LIN {X 0,Y 115.598,Z 257.735,A -85,B 0,C 180,E1 -25782.895,E2 -25782.895} C_VEL
LIN {X 0,Y 117.67,Z 260.063,A -85,B 0,C 180,E1 -25784.586,E2 -25784.586} C_VEL
LIN {X 0,Y 118.631,Z 260.945,A -85,B 0,C 180,E1 -25785.308,E2 -25785.308} C_VEL
LIN {X 0,Y 120.566,Z 264.086,A -85,B 0,C 180,E1 -25786.824,E2 -25786.824} C_VEL
LIN {X 0,Y 122.311,Z 266.016,A -85,B 0,C 180,E1 -25788.026,E2 -25788.026} C_VEL
LIN {X 0,Y 125.956,Z 271.384,A -85,B 0,C 180,E1 -25790.457,E2 -25790.457} C_VEL
LIN {X 0,Y 130.306,Z 277.986,A -85,B 0,C 180,E1 -25793.063,E2 -25793.063} C_VEL
LIN {X 0,Y 136.455,Z 288.82,A -85,B 0,C 180,E1 -25796.428,E2 -25796.428} C_VEL
LIN {X 0,Y 142.566,Z 302.152,A -85,B 0,C 180,E1 -25799.513,E2 -25799.513} C_VEL
LIN {X 0,Y 139.129,Z 349.924,A -85,B 0,C 180,E1 -25801.622,E2 -25801.622} C_VEL
LIN {X 0,Y 137.337,Z 363.693,A -85,B 0,C 180,E1 -25802.791,E2 -25802.791} C_VEL
LIN {X 0,Y 135.158,Z 375.917,A -85,B 0,C 180,E1 -25804.399,E2 -25804.399} C_VEL
LIN {X 0,Y 132.259,Z 387.767,A -85,B 0,C 180,E1 -25806.521,E2 -25806.521} C_VEL
LIN {X 0,Y 128.943,Z 399.162,A -85,B 0,C 180,E1 -25809.258,E2 -25809.258} C_VEL
LIN {X 0,Y 125.816,Z 408.801,A -85,B 0,C 180,E1 -25812.288,E2 -25812.288} C_VEL
LIN {X 0,Y 122.59,Z 417.663,A -85,B 0,C 180,E1 -25815.82,E2 -25815.82} C_VEL
LIN {X 0,Y 118.993,Z 426.966,A -85,B 0,C 180,E1 -25820.659,E2 -25820.659} C_VEL
LIN {X 0,Y 116.23,Z 434.328,A -85,B 0,C 180,E1 -25825.672,E2 -25825.672} C_VEL
LIN {X 0,Y 114.556,Z 439.301,A -85,B 0,C 180,E1 -25830.006,E2 -25830.006} C_VEL
LIN {X 0,Y 113.016,Z 444.479,A -85,B 0,C 180,E1 -25835.755,E2 -25835.755} C_VEL
LIN {X 0,Y 112.2,Z 447.894,A -85,B 0,C 180,E1 -25840.836,E2 -25840.836} C_VEL
LIN {X 0,Y 112.013,Z 449.826,A -85,B 0,C 180,E1 -25844.54,E2 -25844.54} C_VEL
LIN {X 0,Y 112.506,Z 451.951,A -85,B 0,C 180,E1 -25850.447,E2 -25850.447} C_VEL
LIN {X 0,Y 113.673,Z 452.945,A -85,B 0,C 180,E1 -25855.649,E2 -25855.649} C_VEL
LIN {X 0,Y 116.312,Z 452.961,A -85,B 0,C 180,E1 -25862.23,E2 -25862.23} C_VEL
LIN {X 0,Y 118.692,Z 452.233,A -85,B 0,C 180,E1 -25866.311,E2 -25866.311} C_VEL
LIN {X 0,Y 123.419,Z 449.925,A -85,B 0,C 180,E1 -25872.247,E2 -25872.247} C_VEL
LIN {X 0,Y 128.871,Z 446.362,A -85,B 0,C 180,E1 -25877.413,E2 -25877.413} C_VEL
LIN {X 0,Y 134.492,Z 441.991,A -85,B 0,C 180,E1 -25881.615,E2 -25881.615} C_VEL
LIN {X 0,Y 140.722,Z 436.325,A -85,B 0,C 180,E1 -25885.493,E2 -25885.493} C_VEL
LIN {X 0,Y 147.535,Z 429.154,A -85,B 0,C 180,E1 -25889.032,E2 -25889.032} C_VEL
LIN {X 0,Y 154.85,Z 420.055,A -85,B 0,C 180,E1 -25892.254,E2 -25892.254} C_VEL
LIN {X 0,Y 161.376,Z 410.613,A -85,B 0,C 180,E1 -25894.678,E2 -25894.678} C_VEL
LIN {X 0,Y 167.361,Z 400.08,A -85,B 0,C 180,E1 -25896.72,E2 -25896.72} C_VEL
LIN {X 0,Y 172.914,Z 387.981,A -85,B 0,C 180,E1 -25898.493,E2 -25898.493} C_VEL
LIN {X 0,Y 176.998,Z 376.677,A -85,B 0,C 180,E1 -25899.727,E2 -25899.727} C_VEL
LIN {X 0,Y 180.453,Z 363.897,A -85,B 0,C 180,E1 -25900.713,E2 -25900.713} C_VEL
LIN {X 0,Y 182.767,Z 351.132,A -85,B 0,C 180,E1 -25901.395,E2 -25901.395} C_VEL
LIN {X 0,Y 184.15,Z 337.384,A -85,B 0,C 180,E1 -25901.89,E2 -25901.89} C_VEL
LIN {X 0,Y 180.509,Z 329.961,A -85,B 0,C 180,E1 -25905.125,E2 -25905.125} C_VEL
LIN {X 0,Y 177.491,Z 324.525,A -85,B 0,C 180,E1 -25908.22,E2 -25908.22} C_VEL
LIN {X 0,Y 175.588,Z 321.158,A -85,B 0,C 180,E1 -25910.497,E2 -25910.497} C_VEL
LIN {X 0,Y 173.971,Z 318.349,A -85,B 0,C 180,E1 -25912.748,E2 -25912.748} C_VEL
LIN {X 0,Y 172.019,Z 314.67,A -85,B 0,C 180,E1 -25916.245,E2 -25916.245} C_VEL
LIN {X 0,Y 170.224,Z 311.982,A -85,B 0,C 180,E1 -25920.807,E2 -25920.807} C_VEL
LIN {X 0,Y 169.821,Z 310.313,A -85,B 0,C 180,E1 -25922.93,E2 -25922.93} C_VEL
LIN {X 0,Y 169.608,Z 310.274,A -85,B 0,C 180,E1 -25930.406,E2 -25930.406} C_VEL
LIN {X 0,Y 171.721,Z 314.762,A -85,B 0,C 180,E1 -25937.684,E2 -25937.684} C_VEL
LIN {X 0,Y 172.317,Z 315.843,A -85,B 0,C 180,E1 -25938.909,E2 -25938.909} C_VEL
LIN {X 0,Y 174.722,Z 321.19,A -85,B 0,C 180,E1 -25942.984,E2 -25942.984} C_VEL
LIN {X 0,Y 177.011,Z 326.343,A -85,B 0,C 180,E1 -25945.976,E2 -25945.976} C_VEL
LIN {X 0,Y 180.16,Z 334.211,A -85,B 0,C 180,E1 -25949.464,E2 -25949.464} C_VEL
LIN {X 0,Y 182.891,Z 341.732,A -85,B 0,C 180,E1 -25952.106,E2 -25952.106} C_VEL
LIN {X 0,Y 183.682,Z 344.092,A -85,B 0,C 180,E1 -25952.827,E2 -25952.827} C_VEL
LIN {X 0,Y 181.815,Z 360.999,A -85,B 0,C 180,E1 -25953.403,E2 -25953.403} C_VEL
LIN {X 0,Y 179.086,Z 374.216,A -85,B 0,C 180,E1 -25954.07,E2 -25954.07} C_VEL
LIN {X 0,Y 175.617,Z 385.637,A -85,B 0,C 180,E1 -25954.877,E2 -25954.877} C_VEL
LIN {X 0,Y 170.745,Z 398.004,A -85,B 0,C 180,E1 -25956.12,E2 -25956.12} C_VEL
LIN {X 0,Y 165.285,Z 409.082,A -85,B 0,C 180,E1 -25957.632,E2 -25957.632} C_VEL
LIN {X 0,Y 160.004,Z 418.068,A -85,B 0,C 180,E1 -25959.271,E2 -25959.271} C_VEL
LIN {X 0,Y 154.247,Z 426.49,A -85,B 0,C 180,E1 -25961.253,E2 -25961.253} C_VEL
LIN {X 0,Y 146.992,Z 435.652,A -85,B 0,C 180,E1 -25964.176,E2 -25964.176} C_VEL
LIN {X 0,Y 140.246,Z 443.059,A -85,B 0,C 180,E1 -25967.427,E2 -25967.427} C_VEL
LIN {X 0,Y 133.984,Z 449.038,A -85,B 0,C 180,E1 -25970.988,E2 -25970.988} C_VEL
LIN {X 0,Y 127.732,Z 454.471,A -85,B 0,C 180,E1 -25975.623,E2 -25975.623} C_VEL
LIN {X 0,Y 123.721,Z 457.472,A -85,B 0,C 180,E1 -25979.25,E2 -25979.25} C_VEL
LIN {X 0,Y 120.835,Z 459.395,A -85,B 0,C 180,E1 -25982.267,E2 -25982.267} C_VEL
LIN {X 0,Y 118.413,Z 460.88,A -85,B 0,C 180,E1 -25985.448,E2 -25985.448} C_VEL
LIN {X 0,Y 114.715,Z 462.66,A -85,B 0,C 180,E1 -25992.157,E2 -25992.157} C_VEL
LIN {X 0,Y 112.824,Z 462.938,A -85,B 0,C 180,E1 -25999.224,E2 -25999.224} C_VEL
LIN {X 0,Y 112.457,Z 461.612,A -85,B 0,C 180,E1 -26006.411,E2 -26006.411} C_VEL
LIN {X 0,Y 112.608,Z 460.355,A -85,B 0,C 180,E1 -26009.994,E2 -26009.994} C_VEL
LIN {X 0,Y 112.454,Z 457.57,A -85,B 0,C 180,E1 -26015.372,E2 -26015.372} C_VEL
LIN {X 0,Y 112.845,Z 453.713,A -85,B 0,C 180,E1 -26020.761,E2 -26020.761} C_VEL
LIN {X 0,Y 113.912,Z 448.68,A -85,B 0,C 180,E1 -26026.111,E2 -26026.111} C_VEL
LIN {X 0,Y 116.048,Z 442.355,A -85,B 0,C 180,E1 -26031.299,E2 -26031.299} C_VEL
LIN {X 0,Y 118.887,Z 434.38,A -85,B 0,C 180,E1 -26036.309,E2 -26036.309} C_VEL
LIN {X 0,Y 120.485,Z 429.555,A -85,B 0,C 180,E1 -26038.807,E2 -26038.807} C_VEL
LIN {X 0,Y 123.338,Z 422.512,A -85,B 0,C 180,E1 -26041.798,E2 -26041.798} C_VEL
LIN {X 0,Y 126.977,Z 411.905,A -85,B 0,C 180,E1 -26045.405,E2 -26045.405} C_VEL
LIN {X 0,Y 127.946,Z 407.114,A -85,B 0,C 180,E1 -26046.91,E2 -26046.91} C_VEL
LIN {X 0,Y 128.082,Z 399.013,A -85,B 0,C 180,E1 -26049.477,E2 -26049.477} C_VEL
LIN {X 0,Y 128.091,Z 390.513,A -85,B 0,C 180,E1 -26051.766,E2 -26051.766} C_VEL
LIN {X 0,Y 128.802,Z 385.101,A -85,B 0,C 180,E1 -26052.785,E2 -26052.785} C_VEL
LIN {X 0,Y 131.483,Z 371.951,A -85,B 0,C 180,E1 -26054.408,E2 -26054.408} C_VEL
LIN {X 0,Y 133.299,Z 359.02,A -85,B 0,C 180,E1 -26055.451,E2 -26055.451} C_VEL
LIN {X 0,Y 135.911,Z 320.414,A -85,B 0,C 180,E1 -26057.292,E2 -26057.292} C_VEL
LIN {X 0,Y 135.134,Z 306.061,A -85,B 0,C 180,E1 -26058.586,E2 -26058.586} C_VEL
LIN {X 0,Y 131.253,Z 294.436,A -85,B 0,C 180,E1 -26060.995,E2 -26060.995} C_VEL
LIN {X 0,Y 126.575,Z 283.308,A -85,B 0,C 180,E1 -26063.984,E2 -26063.984} C_VEL
LIN {X 0,Y 121.024,Z 274.535,A -85,B 0,C 180,E1 -26067.662,E2 -26067.662} C_VEL
LIN {X 0,Y 118.107,Z 270.401,A -85,B 0,C 180,E1 -26069.818,E2 -26069.818} C_VEL
LIN {X 0,Y 115.689,Z 266.882,A -85,B 0,C 180,E1 -26071.789,E2 -26071.789} C_VEL
LIN {X 0,Y 112.936,Z 263.653,A -85,B 0,C 180,E1 -26074.175,E2 -26074.175} C_VEL
LIN {X 0,Y 111.942,Z 261.643,A -85,B 0,C 180,E1 -26075.207,E2 -26075.207} C_VEL
LIN {X 0,Y 109.374,Z 259.576,A -85,B 0,C 180,E1 -26077.695,E2 -26077.695} C_VEL
LIN {X 0,Y 108.072,Z 256.993,A -85,B 0,C 180,E1 -26079.291,E2 -26079.291} C_VEL
LIN {X 0,Y 107.89,Z 256.04,A -85,B 0,C 180,E1 -26079.752,E2 -26079.752} C_VEL
LIN {X 0,Y 108.176,Z 255.998,A -85,B 0,C 180,E1 -26086.987,E2 -26086.987} C_VEL
LIN {X 0,Y 108.295,Z 255.994,A -85,B 0,C 180,E1 -26092.541,E2 -26092.541} C_VEL
LIN {X 0,Y 108.858,Z 255.852,A -85,B 0,C 180,E1 -26099.999,E2 -26099.999} C_VEL
LIN {X 0,Y 108.268,Z 255.998,A -85,B 0,C 180,E1 -26107.458,E2 -26107.458} C_VEL
LIN {X 0,Y 108.114,Z 256.003,A -85,B 0,C 180,E1 -26112.871,E2 -26112.871} C_VEL
LIN {X 0,Y 107.838,Z 256.033,A -85,B 0,C 180,E1 -26119.016,E2 -26119.016} C_VEL
LIN {X 0,Y 107.795,Z 256.055,A -85,B 0,C 180,E1 -26124.136,E2 -26124.136} C_VEL
LIN {X 0,Y 107.756,Z 255.999,A -85,B 0,C 180,E1 -26132.039,E2 -26132.039} C_VEL
LIN {X 0,Y 107.702,Z 256.263,A -85,B 0,C 180,E1 -26135.963,E2 -26135.963} C_VEL
LIN {X 0,Y 108.55,Z 258.612,A -85,B 0,C 180,E1 -26137.128,E2 -26137.128} C_VEL
LIN {X 0,Y 110.505,Z 260.866,A -85,B 0,C 180,E1 -26139.223,E2 -26139.223} C_VEL
LIN {X 0,Y 111.899,Z 261.779,A -85,B 0,C 180,E1 -26140.516,E2 -26140.516} C_VEL
LIN {X 0,Y 113.733,Z 264.939,A -85,B 0,C 180,E1 -26142.326,E2 -26142.326} C_VEL
LIN {X 0,Y 115.758,Z 267.201,A -85,B 0,C 180,E1 -26144.038,E2 -26144.038} C_VEL
LIN {X 0,Y 118.436,Z 270.876,A -85,B 0,C 180,E1 -26146.181,E2 -26146.181} C_VEL
LIN {X 0,Y 122.217,Z 276.39,A -85,B 0,C 180,E1 -26148.922,E2 -26148.922} C_VEL
LIN {X 0,Y 127.209,Z 284.367,A -85,B 0,C 180,E1 -26152.151,E2 -26152.151} C_VEL
LIN {X 0,Y 132.861,Z 294.969,A -85,B 0,C 180,E1 -26155.449,E2 -26155.449} C_VEL
LIN {X 0,Y 136.897,Z 304.064,A -85,B 0,C 180,E1 -26157.667,E2 -26157.667} C_VEL
LIN {X 0,Y 133.557,Z 350.059,A -85,B 0,C 180,E1 -26159.779,E2 -26159.779} C_VEL
LIN {X 0,Y 131.734,Z 363.498,A -85,B 0,C 180,E1 -26160.93,E2 -26160.93} C_VEL
LIN {X 0,Y 129.484,Z 375.625,A -85,B 0,C 180,E1 -26162.534,E2 -26162.534} C_VEL
LIN {X 0,Y 126.733,Z 386.809,A -85,B 0,C 180,E1 -26164.555,E2 -26164.555} C_VEL
LIN {X 0,Y 123.531,Z 397.171,A -85,B 0,C 180,E1 -26166.983,E2 -26166.983} C_VEL
LIN {X 0,Y 120.233,Z 407.16,A -85,B 0,C 180,E1 -26170.094,E2 -26170.094} C_VEL
LIN {X 0,Y 116.295,Z 417.47,A -85,B 0,C 180,E1 -26174.228,E2 -26174.228} C_VEL
LIN {X 0,Y 113.089,Z 425.367,A -85,B 0,C 180,E1 -26178.355,E2 -26178.355} C_VEL
LIN {X 0,Y 109.981,Z 433.068,A -85,B 0,C 180,E1 -26183.586,E2 -26183.586} C_VEL
LIN {X 0,Y 108.017,Z 438.34,A -85,B 0,C 180,E1 -26188.142,E2 -26188.142} C_VEL
LIN {X 0,Y 106.33,Z 443.457,A -85,B 0,C 180,E1 -26193.796,E2 -26193.796} C_VEL
LIN {X 0,Y 105.237,Z 447.449,A -85,B 0,C 180,E1 -26199.617,E2 -26199.617} C_VEL
LIN {X 0,Y 104.946,Z 450.389,A -85,B 0,C 180,E1 -26205.543,E2 -26205.543} C_VEL
LIN {X 0,Y 105.491,Z 452.26,A -85,B 0,C 180,E1 -26211.143,E2 -26211.143} C_VEL
LIN {X 0,Y 107.022,Z 453.33,A -85,B 0,C 180,E1 -26217.371,E2 -26217.371} C_VEL
LIN {X 0,Y 109.686,Z 453.312,A -85,B 0,C 180,E1 -26223.598,E2 -26223.598} C_VEL
LIN {X 0,Y 112.771,Z 452.443,A -85,B 0,C 180,E1 -26228.554,E2 -26228.554} C_VEL
LIN {X 0,Y 117.389,Z 450.323,A -85,B 0,C 180,E1 -26234.076,E2 -26234.076} C_VEL
LIN {X 0,Y 123.944,Z 446.316,A -85,B 0,C 180,E1 -26239.953,E2 -26239.953} C_VEL
LIN {X 0,Y 129.989,Z 441.835,A -85,B 0,C 180,E1 -26244.195,E2 -26244.195} C_VEL
LIN {X 0,Y 136.662,Z 436.053,A -85,B 0,C 180,E1 -26248.053,E2 -26248.053} C_VEL
LIN {X 0,Y 143.881,Z 428.685,A -85,B 0,C 180,E1 -26251.549,E2 -26251.549} C_VEL
LIN {X 0,Y 150.23,Z 421.102,A -85,B 0,C 180,E1 -26254.23,E2 -26254.23} C_VEL
LIN {X 0,Y 156.948,Z 411.855,A -85,B 0,C 180,E1 -26256.627,E2 -26256.627} C_VEL
LIN {X 0,Y 163.162,Z 401.546,A -85,B 0,C 180,E1 -26258.664,E2 -26258.664} C_VEL
LIN {X 0,Y 168.883,Z 389.773,A -85,B 0,C 180,E1 -26260.389,E2 -26260.389} C_VEL
LIN {X 0,Y 173.476,Z 377.761,A -85,B 0,C 180,E1 -26261.714,E2 -26261.714} C_VEL
LIN {X 0,Y 177.043,Z 365.385,A -85,B 0,C 180,E1 -26262.664,E2 -26262.664} C_VEL
LIN {X 0,Y 179.577,Z 352.18,A -85,B 0,C 180,E1 -26263.381,E2 -26263.381} C_VEL
LIN {X 0,Y 180.823,Z 341.143,A -85,B 0,C 180,E1 -26263.779,E2 -26263.779} C_VEL
LIN {X 0,Y 177.84,Z 334.851,A -85,B 0,C 180,E1 -26266.721,E2 -26266.721} C_VEL
LIN {X 0,Y 174.43,Z 328.348,A -85,B 0,C 180,E1 -26270.726,E2 -26270.726} C_VEL
LIN {X 0,Y 172.539,Z 324.937,A -85,B 0,C 180,E1 -26273.503,E2 -26273.503} C_VEL
LIN {X 0,Y 170.819,Z 321.538,A -85,B 0,C 180,E1 -26276.809,E2 -26276.809} C_VEL
LIN {X 0,Y 169.114,Z 318.519,A -85,B 0,C 180,E1 -26281.705,E2 -26281.705} C_VEL
LIN {X 0,Y 168.905,Z 317.431,A -85,B 0,C 180,E1 -26283.029,E2 -26283.029} C_VEL
LIN {X 0,Y 168.609,Z 317.256,A -85,B 0,C 180,E1 -26289.598,E2 -26289.598} C_VEL
LIN {X 0,Y 168.744,Z 317.561,A -85,B 0,C 180,E1 -26290.678,E2 -26290.678} C_VEL
LIN {X 0,Y 170.54,Z 321.593,A -85,B 0,C 180,E1 -26297.114,E2 -26297.114} C_VEL
LIN {X 0,Y 171.05,Z 322.554,A -85,B 0,C 180,E1 -26298.239,E2 -26298.239} C_VEL
LIN {X 0,Y 173.144,Z 327.626,A -85,B 0,C 180,E1 -26302.132,E2 -26302.132} C_VEL
LIN {X 0,Y 175.554,Z 333.434,A -85,B 0,C 180,E1 -26305.491,E2 -26305.491} C_VEL
LIN {X 0,Y 178.666,Z 341.989,A -85,B 0,C 180,E1 -26309.129,E2 -26309.129} C_VEL
LIN {X 0,Y 180.373,Z 347.162,A -85,B 0,C 180,E1 -26310.905,E2 -26310.905} C_VEL
LIN {X 0,Y 178.545,Z 361.926,A -85,B 0,C 180,E1 -26311.402,E2 -26311.402} C_VEL
LIN {X 0,Y 175.581,Z 375.181,A -85,B 0,C 180,E1 -26312.086,E2 -26312.086} C_VEL
LIN {X 0,Y 171.691,Z 387.222,A -85,B 0,C 180,E1 -26312.95,E2 -26312.95} C_VEL
LIN {X 0,Y 166.685,Z 399.203,A -85,B 0,C 180,E1 -26314.162,E2 -26314.162} C_VEL
LIN {X 0,Y 161.069,Z 409.925,A -85,B 0,C 180,E1 -26315.642,E2 -26315.642} C_VEL
LIN {X 0,Y 156.285,Z 417.714,A -85,B 0,C 180,E1 -26317.041,E2 -26317.041} C_VEL
LIN {X 0,Y 149.687,Z 426.975,A -85,B 0,C 180,E1 -26319.222,E2 -26319.222} C_VEL
LIN {X 0,Y 142.151,Z 435.977,A -85,B 0,C 180,E1 -26322.13,E2 -26322.13} C_VEL
LIN {X 0,Y 135.116,Z 443.26,A -85,B 0,C 180,E1 -26325.395,E2 -26325.395} C_VEL
LIN {X 0,Y 128.546,Z 449.131,A -85,B 0,C 180,E1 -26328.996,E2 -26328.996} C_VEL
LIN {X 0,Y 122.587,Z 453.934,A -85,B 0,C 180,E1 -26333.191,E2 -26333.191} C_VEL
LIN {X 0,Y 117.654,Z 457.386,A -85,B 0,C 180,E1 -26337.475,E2 -26337.475} C_VEL
LIN {X 0,Y 114.583,Z 459.254,A -85,B 0,C 180,E1 -26340.61,E2 -26340.61} C_VEL
LIN {X 0,Y 109.712,Z 461.719,A -85,B 0,C 180,E1 -26347.392,E2 -26347.392} C_VEL
LIN {X 0,Y 106.694,Z 462.679,A -85,B 0,C 180,E1 -26354.718,E2 -26354.718} C_VEL
LIN {X 0,Y 105.412,Z 462.047,A -85,B 0,C 180,E1 -26362.331,E2 -26362.331} C_VEL
LIN {X 0,Y 105.481,Z 460.562,A -85,B 0,C 180,E1 -26368.086,E2 -26368.086} C_VEL
LIN {X 0,Y 105.447,Z 459.313,A -85,B 0,C 180,E1 -26371.24,E2 -26371.24} C_VEL
LIN {X 0,Y 105.455,Z 455.795,A -85,B 0,C 180,E1 -26377.652,E2 -26377.652} C_VEL
LIN {X 0,Y 106.132,Z 451.469,A -85,B 0,C 180,E1 -26383.393,E2 -26383.393} C_VEL
LIN {X 0,Y 107.699,Z 445.917,A -85,B 0,C 180,E1 -26389.034,E2 -26389.034} C_VEL
LIN {X 0,Y 110.293,Z 438.971,A -85,B 0,C 180,E1 -26394.459,E2 -26394.459} C_VEL
LIN {X 0,Y 112.957,Z 431.83,A -85,B 0,C 180,E1 -26398.819,E2 -26398.819} C_VEL
LIN {X 0,Y 116.571,Z 423.262,A -85,B 0,C 180,E1 -26402.851,E2 -26402.851} C_VEL
LIN {X 0,Y 120.043,Z 413.778,A -85,B 0,C 180,E1 -26406.343,E2 -26406.343} C_VEL
LIN {X 0,Y 123.985,Z 402.01,A -85,B 0,C 180,E1 -26409.609,E2 -26409.609} C_VEL
LIN {X 0,Y 126.512,Z 394.008,A -85,B 0,C 180,E1 -26411.263,E2 -26411.263} C_VEL
LIN {X 0,Y 128.802,Z 385.101,A -85,B 0,C 180,E1 -26412.785,E2 -26412.785} C_VEL
LIN {X 0,Y 129.472,Z 379.628,A -85,B 0,C 180,E1 -26413.721,E2 -26413.721} C_VEL
LIN {X 0,Y 128.938,Z 370.556,A -85,B 0,C 180,E1 -26415.498,E2 -26415.498} C_VEL
LIN {X 0,Y 128.108,Z 361.329,A -85,B 0,C 180,E1 -26417.066,E2 -26417.066} C_VEL
LIN {X 0,Y 128.167,Z 355.554,A -85,B 0,C 180,E1 -26417.626,E2 -26417.626} C_VEL
LIN {X 0,Y 130.583,Z 321.958,A -85,B 0,C 180,E1 -26419.203,E2 -26419.203} C_VEL
LIN {X 0,Y 129.906,Z 308.256,A -85,B 0,C 180,E1 -26420.512,E2 -26420.512} C_VEL
LIN {X 0,Y 126.572,Z 297.933,A -85,B 0,C 180,E1 -26422.791,E2 -26422.791} C_VEL
LIN {X 0,Y 122.392,Z 287.675,A -85,B 0,C 180,E1 -26425.719,E2 -26425.719} C_VEL
LIN {X 0,Y 116.999,Z 279.06,A -85,B 0,C 180,E1 -26429.652,E2 -26429.652} C_VEL
LIN {X 0,Y 114.998,Z 276.119,A -85,B 0,C 180,E1 -26431.277,E2 -26431.277} C_VEL
LIN {X 0,Y 112.116,Z 272.044,A -85,B 0,C 180,E1 -26433.831,E2 -26433.831} C_VEL
LIN {X 0,Y 109.662,Z 268.586,A -85,B 0,C 180,E1 -26436.266,E2 -26436.266} C_VEL
LIN {X 0,Y 109.026,Z 267.677,A -85,B 0,C 180,E1 -26436.946,E2 -26436.946} C_VEL
LIN {X 0,Y 106.602,Z 265.096,A -85,B 0,C 180,E1 -26439.623,E2 -26439.623} C_VEL
LIN {X 0,Y 105.384,Z 262.679,A -85,B 0,C 180,E1 -26441.279,E2 -26441.279} C_VEL
LIN {X 0,Y 102.98,Z 261.081,A -85,B 0,C 180,E1 -26444.428,E2 -26444.428} C_VEL
LIN {X 0,Y 101.585,Z 258.686,A -85,B 0,C 180,E1 -26446.813,E2 -26446.813} C_VEL
LIN {X 0,Y 101.185,Z 256.865,A -85,B 0,C 180,E1 -26447.972,E2 -26447.972} C_VEL
LIN {X 0,Y 101.236,Z 256.874,A -85,B 0,C 180,E1 -26452.018,E2 -26452.018} C_VEL
LIN {X 0,Y 101.789,Z 256.73,A -85,B 0,C 180,E1 -26459.999,E2 -26459.999} C_VEL
LIN {X 0,Y 101.201,Z 256.877,A -85,B 0,C 180,E1 -26467.982,E2 -26467.982} C_VEL
LIN {X 0,Y 101.027,Z 256.887,A -85,B 0,C 180,E1 -26473.167,E2 -26473.167} C_VEL
LIN {X 0,Y 100.755,Z 256.916,A -85,B 0,C 180,E1 -26480.411,E2 -26480.411} C_VEL
LIN {X 0,Y 100.658,Z 256.936,A -85,B 0,C 180,E1 -26487.127,E2 -26487.127} C_VEL
LIN {X 0,Y 101.31,Z 259.154,A -85,B 0,C 180,E1 -26488.624,E2 -26488.624} C_VEL
LIN {X 0,Y 103.154,Z 261.396,A -85,B 0,C 180,E1 -26491.603,E2 -26491.603} C_VEL
LIN {X 0,Y 105.398,Z 263.032,A -85,B 0,C 180,E1 -26494.525,E2 -26494.525} C_VEL
LIN {X 0,Y 107.216,Z 266.21,A -85,B 0,C 180,E1 -26496.887,E2 -26496.887} C_VEL
LIN {X 0,Y 109.419,Z 268.263,A -85,B 0,C 180,E1 -26499.22,E2 -26499.22} C_VEL
LIN {X 0,Y 111.76,Z 271.758,A -85,B 0,C 180,E1 -26501.598,E2 -26501.598} C_VEL
LIN {X 0,Y 113.194,Z 273.656,A -85,B 0,C 180,E1 -26502.909,E2 -26502.909} C_VEL
LIN {X 0,Y 116.595,Z 278.511,A -85,B 0,C 180,E1 -26505.775,E2 -26505.775} C_VEL
LIN {X 0,Y 120.729,Z 284.861,A -85,B 0,C 180,E1 -26508.868,E2 -26508.868} C_VEL
LIN {X 0,Y 125.575,Z 293.525,A -85,B 0,C 180,E1 -26512.126,E2 -26512.126} C_VEL
LIN {X 0,Y 129.592,Z 301.854,A -85,B 0,C 180,E1 -26514.602,E2 -26514.602} C_VEL
LIN {X 0,Y 131.485,Z 306.259,A -85,B 0,C 180,E1 -26515.728,E2 -26515.728} C_VEL
LIN {X 0,Y 128.149,Z 350.109,A -85,B 0,C 180,E1 -26517.774,E2 -26517.774} C_VEL
LIN {X 0,Y 126.207,Z 363.77,A -85,B 0,C 180,E1 -26518.958,E2 -26518.958} C_VEL
LIN {X 0,Y 123.725,Z 376.39,A -85,B 0,C 180,E1 -26520.674,E2 -26520.674} C_VEL
LIN {X 0,Y 120.822,Z 387.463,A -85,B 0,C 180,E1 -26522.746,E2 -26522.746} C_VEL
LIN {X 0,Y 117.461,Z 397.763,A -85,B 0,C 180,E1 -26525.248,E2 -26525.248} C_VEL
LIN {X 0,Y 113.641,Z 408.566,A -85,B 0,C 180,E1 -26528.79,E2 -26528.79} C_VEL
LIN {X 0,Y 110.179,Z 417.08,A -85,B 0,C 180,E1 -26532.371,E2 -26532.371} C_VEL
LIN {X 0,Y 106.736,Z 425.102,A -85,B 0,C 180,E1 -26536.684,E2 -26536.684} C_VEL
LIN {X 0,Y 103.351,Z 432.944,A -85,B 0,C 180,E1 -26542.191,E2 -26542.191} C_VEL
LIN {X 0,Y 100.826,Z 439.224,A -85,B 0,C 180,E1 -26548.01,E2 -26548.01} C_VEL
LIN {X 0,Y 99.105,Z 444.228,A -85,B 0,C 180,E1 -26554.073,E2 -26554.073} C_VEL
LIN {X 0,Y 98.044,Z 448.115,A -85,B 0,C 180,E1 -26560.33,E2 -26560.33} C_VEL
LIN {X 0,Y 97.895,Z 450.952,A -85,B 0,C 180,E1 -26566.694,E2 -26566.694} C_VEL
LIN {X 0,Y 98.509,Z 452.573,A -85,B 0,C 180,E1 -26571.96,E2 -26571.96} C_VEL
LIN {X 0,Y 100.475,Z 453.697,A -85,B 0,C 180,E1 -26579.321,E2 -26579.321} C_VEL
LIN {X 0,Y 103.15,Z 453.662,A -85,B 0,C 180,E1 -26585.157,E2 -26585.157} C_VEL
LIN {X 0,Y 107.033,Z 452.62,A -85,B 0,C 180,E1 -26591.047,E2 -26591.047} C_VEL
LIN {X 0,Y 111.519,Z 450.723,A -85,B 0,C 180,E1 -26596.115,E2 -26596.115} C_VEL
LIN {X 0,Y 117.275,Z 447.548,A -85,B 0,C 180,E1 -26601.177,E2 -26601.177} C_VEL
LIN {X 0,Y 123.808,Z 443.141,A -85,B 0,C 180,E1 -26605.75,E2 -26605.75} C_VEL
LIN {X 0,Y 131.651,Z 436.827,A -85,B 0,C 180,E1 -26610.169,E2 -26610.169} C_VEL
LIN {X 0,Y 137.869,Z 430.918,A -85,B 0,C 180,E1 -26613.133,E2 -26613.133} C_VEL
LIN {X 0,Y 144.45,Z 423.759,A -85,B 0,C 180,E1 -26615.818,E2 -26615.818} C_VEL
LIN {X 0,Y 151.352,Z 415.057,A -85,B 0,C 180,E1 -26618.232,E2 -26618.232} C_VEL
LIN {X 0,Y 157.727,Z 405.372,A -85,B 0,C 180,E1 -26620.268,E2 -26620.268} C_VEL
LIN {X 0,Y 163.731,Z 394.313,A -85,B 0,C 180,E1 -26622.017,E2 -26622.017} C_VEL
LIN {X 0,Y 168.686,Z 382.924,A -85,B 0,C 180,E1 -26623.382,E2 -26623.382} C_VEL
LIN {X 0,Y 172.688,Z 370.99,A -85,B 0,C 180,E1 -26624.411,E2 -26624.411} C_VEL
LIN {X 0,Y 175.86,Z 357.568,A -85,B 0,C 180,E1 -26625.242,E2 -26625.242} C_VEL
LIN {X 0,Y 177.67,Z 344.898,A -85,B 0,C 180,E1 -26625.76,E2 -26625.76} C_VEL
LIN {X 0,Y 175.012,Z 339.21,A -85,B 0,C 180,E1 -26628.711,E2 -26628.711} C_VEL
LIN {X 0,Y 172.407,Z 334.063,A -85,B 0,C 180,E1 -26632.167,E2 -26632.167} C_VEL
LIN {X 0,Y 171.041,Z 331.341,A -85,B 0,C 180,E1 -26634.443,E2 -26634.443} C_VEL
LIN {X 0,Y 169.529,Z 328.25,A -85,B 0,C 180,E1 -26637.625,E2 -26637.625} C_VEL
LIN {X 0,Y 168.05,Z 325.135,A -85,B 0,C 180,E1 -26642.559,E2 -26642.559} C_VEL
LIN {X 0,Y 167.929,Z 324.429,A -85,B 0,C 180,E1 -26643.485,E2 -26643.485} C_VEL
LIN {X 0,Y 167.787,Z 324.376,A -85,B 0,C 180,E1 -26650.083,E2 -26650.083} C_VEL
LIN {X 0,Y 169.424,Z 328.465,A -85,B 0,C 180,E1 -26656.643,E2 -26656.643} C_VEL
LIN {X 0,Y 169.908,Z 329.621,A -85,B 0,C 180,E1 -26657.824,E2 -26657.824} C_VEL
LIN {X 0,Y 171.568,Z 333.93,A -85,B 0,C 180,E1 -26661.174,E2 -26661.174} C_VEL
LIN {X 0,Y 173.68,Z 339.465,A -85,B 0,C 180,E1 -26664.426,E2 -26664.426} C_VEL
LIN {X 0,Y 176.636,Z 348.336,A -85,B 0,C 180,E1 -26668.196,E2 -26668.196} C_VEL
LIN {X 0,Y 177.235,Z 350.361,A -85,B 0,C 180,E1 -26668.897,E2 -26668.897} C_VEL
LIN {X 0,Y 175.421,Z 363.199,A -85,B 0,C 180,E1 -26669.363,E2 -26669.363} C_VEL
LIN {X 0,Y 172.286,Z 376.213,A -85,B 0,C 180,E1 -26670.037,E2 -26670.037} C_VEL
LIN {X 0,Y 167.967,Z 388.806,A -85,B 0,C 180,E1 -26670.936,E2 -26670.936} C_VEL
LIN {X 0,Y 162.83,Z 400.288,A -85,B 0,C 180,E1 -26672.109,E2 -26672.109} C_VEL
LIN {X 0,Y 156.333,Z 411.904,A -85,B 0,C 180,E1 -26673.729,E2 -26673.729} C_VEL
LIN {X 0,Y 149.389,Z 422.229,A -85,B 0,C 180,E1 -26675.754,E2 -26675.754} C_VEL
LIN {X 0,Y 142.631,Z 430.627,A -85,B 0,C 180,E1 -26677.964,E2 -26677.964} C_VEL
LIN {X 0,Y 134.997,Z 438.85,A -85,B 0,C 180,E1 -26680.984,E2 -26680.984} C_VEL
LIN {X 0,Y 127.788,Z 445.509,A -85,B 0,C 180,E1 -26684.357,E2 -26684.357} C_VEL
LIN {X 0,Y 121.153,Z 450.854,A -85,B 0,C 180,E1 -26688.153,E2 -26688.153} C_VEL
LIN {X 0,Y 115.273,Z 455.058,A -85,B 0,C 180,E1 -26692.43,E2 -26692.43} C_VEL
LIN {X 0,Y 111.713,Z 457.31,A -85,B 0,C 180,E1 -26695.51,E2 -26695.51} C_VEL
LIN {X 0,Y 108.44,Z 459.097,A -85,B 0,C 180,E1 -26698.765,E2 -26698.765} C_VEL
LIN {X 0,Y 103.185,Z 461.483,A -85,B 0,C 180,E1 -26705.874,E2 -26705.874} C_VEL
LIN {X 0,Y 101.215,Z 462.111,A -85,B 0,C 180,E1 -26709.68,E2 -26709.68} C_VEL
LIN {X 0,Y 99.818,Z 462.342,A -85,B 0,C 180,E1 -26713.637,E2 -26713.637} C_VEL
LIN {X 0,Y 98.356,Z 461.627,A -85,B 0,C 180,E1 -26721.777,E2 -26721.777} C_VEL
LIN {X 0,Y 98.303,Z 460.702,A -85,B 0,C 180,E1 -26725.893,E2 -26725.893} C_VEL
LIN {X 0,Y 98.397,Z 459.162,A -85,B 0,C 180,E1 -26730.452,E2 -26730.452} C_VEL
LIN {X 0,Y 98.312,Z 456.424,A -85,B 0,C 180,E1 -26736.148,E2 -26736.148} C_VEL
LIN {X 0,Y 98.856,Z 452.398,A -85,B 0,C 180,E1 -26742.306,E2 -26742.306} C_VEL
LIN {X 0,Y 100.583,Z 446.146,A -85,B 0,C 180,E1 -26749.375,E2 -26749.375} C_VEL
LIN {X 0,Y 103.299,Z 439.327,A -85,B 0,C 180,E1 -26755.155,E2 -26755.155} C_VEL
LIN {X 0,Y 106.125,Z 432.333,A -85,B 0,C 180,E1 -26759.77,E2 -26759.77} C_VEL
LIN {X 0,Y 109.851,Z 423.944,A -85,B 0,C 180,E1 -26764.03,E2 -26764.03} C_VEL
LIN {X 0,Y 113.489,Z 414.728,A -85,B 0,C 180,E1 -26767.688,E2 -26767.688} C_VEL
LIN {X 0,Y 117.166,Z 404.716,A -85,B 0,C 180,E1 -26770.704,E2 -26770.704} C_VEL
LIN {X 0,Y 120.704,Z 393.835,A -85,B 0,C 180,E1 -26773.156,E2 -26773.156} C_VEL
LIN {X 0,Y 123.798,Z 381.791,A -85,B 0,C 180,E1 -26775.191,E2 -26775.191} C_VEL
LIN {X 0,Y 126.391,Z 369.287,A -85,B 0,C 180,E1 -26776.627,E2 -26776.627} C_VEL
LIN {X 0,Y 128.074,Z 356.765,A -85,B 0,C 180,E1 -26777.556,E2 -26777.556} C_VEL
LIN {X 0,Y 128.167,Z 355.554,A -85,B 0,C 180,E1 -26777.626,E2 -26777.626} C_VEL
LIN {X 0,Y 128.101,Z 349.753,A -85,B 0,C 180,E1 -26778.137,E2 -26778.137} C_VEL
LIN {X 0,Y 125.257,Z 330.993,A -85,B 0,C 180,E1 -26780.748,E2 -26780.748} C_VEL
LIN {X 0,Y 125.24,Z 325.177,A -85,B 0,C 180,E1 -26781.209,E2 -26781.209} C_VEL
LIN {X 0,Y 125.244,Z 318.245,A -85,B 0,C 180,E1 -26781.761,E2 -26781.761} C_VEL
LIN {X 0,Y 124.83,Z 310.569,A -85,B 0,C 180,E1 -26782.571,E2 -26782.571} C_VEL
LIN {X 0,Y 121.805,Z 300.833,A -85,B 0,C 180,E1 -26784.871,E2 -26784.871} C_VEL
LIN {X 0,Y 118.355,Z 292.13,A -85,B 0,C 180,E1 -26787.552,E2 -26787.552} C_VEL
LIN {X 0,Y 113.779,Z 284.565,A -85,B 0,C 180,E1 -26791.217,E2 -26791.217} C_VEL
LIN {X 0,Y 111.527,Z 281.154,A -85,B 0,C 180,E1 -26793.229,E2 -26793.229} C_VEL
LIN {X 0,Y 109.219,Z 277.78,A -85,B 0,C 180,E1 -26795.484,E2 -26795.484} C_VEL
LIN {X 0,Y 106.512,Z 273.841,A -85,B 0,C 180,E1 -26798.466,E2 -26798.466} C_VEL
LIN {X 0,Y 104.12,Z 270.857,A -85,B 0,C 180,E1 -26801.426,E2 -26801.426} C_VEL
LIN {X 0,Y 103.232,Z 269.229,A -85,B 0,C 180,E1 -26802.721,E2 -26802.721} C_VEL
LIN {X 0,Y 100.843,Z 267.135,A -85,B 0,C 180,E1 -26806.229,E2 -26806.229} C_VEL
LIN {X 0,Y 99.487,Z 264.386,A -85,B 0,C 180,E1 -26808.926,E2 -26808.926} C_VEL
LIN {X 0,Y 99.089,Z 263.664,A -85,B 0,C 180,E1 -26809.785,E2 -26809.785} C_VEL
LIN {X 0,Y 96.255,Z 261.699,A -85,B 0,C 180,E1 -26816.86,E2 -26816.86} C_VEL
LIN {X 0,Y 95.586,Z 260.24,A -85,B 0,C 180,E1 -26819.999,E2 -26819.999} C_VEL
LIN {X 0,Y 94.765,Z 259.92,A -85,B 0,C 180,E1 -26828.529,E2 -26828.529} C_VEL
LIN {X 0,Y 95.147,Z 261.007,A -85,B 0,C 180,E1 -26833.997,E2 -26833.997} C_VEL
LIN {X 0,Y 98.416,Z 263.644,A -85,B 0,C 180,E1 -26844.702,E2 -26844.702} C_VEL
LIN {X 0,Y 98.947,Z 263.981,A -85,B 0,C 180,E1 -26845.787,E2 -26845.787} C_VEL
LIN {X 0,Y 100.166,Z 266.615,A -85,B 0,C 180,E1 -26848.41,E2 -26848.41} C_VEL
LIN {X 0,Y 103.267,Z 269.57,A -85,B 0,C 180,E1 -26853.131,E2 -26853.131} C_VEL
LIN {X 0,Y 105.569,Z 273.119,A -85,B 0,C 180,E1 -26856.215,E2 -26856.215} C_VEL
LIN {X 0,Y 107.062,Z 274.71,A -85,B 0,C 180,E1 -26857.917,E2 -26857.917} C_VEL
LIN {X 0,Y 110.432,Z 279.633,A -85,B 0,C 180,E1 -26861.476,E2 -26861.476} C_VEL
LIN {X 0,Y 113.826,Z 284.625,A -85,B 0,C 180,E1 -26864.561,E2 -26864.561} C_VEL
LIN {X 0,Y 118.552,Z 292.492,A -85,B 0,C 180,E1 -26868.339,E2 -26868.339} C_VEL
LIN {X 0,Y 123.889,Z 303.026,A -85,B 0,C 180,E1 -26872.104,E2 -26872.104} C_VEL
LIN {X 0,Y 126.196,Z 308.504,A -85,B 0,C 180,E1 -26873.634,E2 -26873.634} C_VEL
LIN {X 0,Y 122.801,Z 350.889,A -85,B 0,C 180,E1 -26875.659,E2 -26875.659} C_VEL
LIN {X 0,Y 120.793,Z 364.168,A -85,B 0,C 180,E1 -26876.83,E2 -26876.83} C_VEL
LIN {X 0,Y 118.107,Z 377.065,A -85,B 0,C 180,E1 -26878.633,E2 -26878.633} C_VEL
LIN {X 0,Y 115.022,Z 388.072,A -85,B 0,C 180,E1 -26880.747,E2 -26880.747} C_VEL
LIN {X 0,Y 111.509,Z 398.315,A -85,B 0,C 180,E1 -26883.326,E2 -26883.326} C_VEL
LIN {X 0,Y 107.545,Z 408.884,A -85,B 0,C 180,E1 -26886.924,E2 -26886.924} C_VEL
LIN {X 0,Y 103.393,Z 418.459,A -85,B 0,C 180,E1 -26891.172,E2 -26891.172} C_VEL
LIN {X 0,Y 99.116,Z 427.662,A -85,B 0,C 180,E1 -26896.685,E2 -26896.685} C_VEL
LIN {X 0,Y 95.748,Z 435.073,A -85,B 0,C 180,E1 -26902.628,E2 -26902.628} C_VEL
LIN {X 0,Y 93.64,Z 440.095,A -85,B 0,C 180,E1 -26907.857,E2 -26907.857} C_VEL
LIN {X 0,Y 91.742,Z 445.529,A -85,B 0,C 180,E1 -26915.215,E2 -26915.215} C_VEL
LIN {X 0,Y 90.86,Z 448.772,A -85,B 0,C 180,E1 -26921.157,E2 -26921.157} C_VEL
LIN {X 0,Y 90.895,Z 451.507,A -85,B 0,C 180,E1 -26928.022,E2 -26928.022} C_VEL
LIN {X 0,Y 91.565,Z 452.883,A -85,B 0,C 180,E1 -26932.923,E2 -26932.923} C_VEL
LIN {X 0,Y 94.06,Z 454.062,A -85,B 0,C 180,E1 -26941.541,E2 -26941.541} C_VEL
LIN {X 0,Y 96.729,Z 454.011,A -85,B 0,C 180,E1 -26946.946,E2 -26946.946} C_VEL
LIN {X 0,Y 101.518,Z 452.793,A -85,B 0,C 180,E1 -26953.816,E2 -26953.816} C_VEL
LIN {X 0,Y 105.83,Z 451.114,A -85,B 0,C 180,E1 -26958.389,E2 -26958.389} C_VEL
LIN {X 0,Y 112.735,Z 447.516,A -85,B 0,C 180,E1 -26964.141,E2 -26964.141} C_VEL
LIN {X 0,Y 119.527,Z 443.164,A -85,B 0,C 180,E1 -26968.564,E2 -26968.564} C_VEL
LIN {X 0,Y 126.827,Z 437.597,A -85,B 0,C 180,E1 -26972.454,E2 -26972.454} C_VEL
LIN {X 0,Y 134.698,Z 430.517,A -85,B 0,C 180,E1 -26975.935,E2 -26975.935} C_VEL
LIN {X 0,Y 141.559,Z 423.19,A -85,B 0,C 180,E1 -26978.573,E2 -26978.573} C_VEL
LIN {X 0,Y 149.491,Z 413.222,A -85,B 0,C 180,E1 -26981.108,E2 -26981.108} C_VEL
LIN {X 0,Y 156.124,Z 403.086,A -85,B 0,C 180,E1 -26983.052,E2 -26983.052} C_VEL
LIN {X 0,Y 162.13,Z 391.796,A -85,B 0,C 180,E1 -26984.648,E2 -26984.648} C_VEL
LIN {X 0,Y 167.172,Z 379.681,A -85,B 0,C 180,E1 -26985.942,E2 -26985.942} C_VEL
LIN {X 0,Y 170.842,Z 368.274,A -85,B 0,C 180,E1 -26986.791,E2 -26986.791} C_VEL
LIN {X 0,Y 173.66,Z 355.622,A -85,B 0,C 180,E1 -26987.502,E2 -26987.502} C_VEL
LIN {X 0,Y 174.651,Z 348.73,A -85,B 0,C 180,E1 -26987.806,E2 -26987.806} C_VEL
LIN {X 0,Y 172.106,Z 343.102,A -85,B 0,C 180,E1 -26991.155,E2 -26991.155} C_VEL
LIN {X 0,Y 169.919,Z 338.362,A -85,B 0,C 180,E1 -26994.77,E2 -26994.77} C_VEL
LIN {X 0,Y 168.376,Z 335.072,A -85,B 0,C 180,E1 -26998.208,E2 -26998.208} C_VEL
LIN {X 0,Y 167.022,Z 331.689,A -85,B 0,C 180,E1 -27003.469,E2 -27003.469} C_VEL
LIN {X 0,Y 166.839,Z 331.331,A -85,B 0,C 180,E1 -27004.834,E2 -27004.834} C_VEL
LIN {X 0,Y 166.867,Z 331.525,A -85,B 0,C 180,E1 -27009.919,E2 -27009.919} C_VEL
LIN {X 0,Y 168.524,Z 335.827,A -85,B 0,C 180,E1 -27016.711,E2 -27016.711} C_VEL
LIN {X 0,Y 170.111,Z 340.422,A -85,B 0,C 180,E1 -27020.323,E2 -27020.323} C_VEL
LIN {X 0,Y 171.862,Z 345.552,A -85,B 0,C 180,E1 -27023.339,E2 -27023.339} C_VEL
LIN {X 0,Y 174.232,Z 353.405,A -85,B 0,C 180,E1 -27026.772,E2 -27026.772} C_VEL
LIN {X 0,Y 173.905,Z 356.707,A -85,B 0,C 180,E1 -27026.962,E2 -27026.962} C_VEL
LIN {X 0,Y 171.079,Z 370.553,A -85,B 0,C 180,E1 -27027.526,E2 -27027.526} C_VEL
LIN {X 0,Y 167.125,Z 383.468,A -85,B 0,C 180,E1 -27028.302,E2 -27028.302} C_VEL
LIN {X 0,Y 162.191,Z 395.316,A -85,B 0,C 180,E1 -27029.303,E2 -27029.303} C_VEL
LIN {X 0,Y 156.217,Z 406.705,A -85,B 0,C 180,E1 -27030.638,E2 -27030.638} C_VEL
LIN {X 0,Y 149.597,Z 417.006,A -85,B 0,C 180,E1 -27032.26,E2 -27032.26} C_VEL
LIN {X 0,Y 142.562,Z 426.272,A -85,B 0,C 180,E1 -27034.335,E2 -27034.335} C_VEL
LIN {X 0,Y 135.739,Z 433.927,A -85,B 0,C 180,E1 -27036.627,E2 -27036.627} C_VEL
LIN {X 0,Y 127.907,Z 441.452,A -85,B 0,C 180,E1 -27039.712,E2 -27039.712} C_VEL
LIN {X 0,Y 120.533,Z 447.536,A -85,B 0,C 180,E1 -27043.207,E2 -27043.207} C_VEL
LIN {X 0,Y 113.792,Z 452.389,A -85,B 0,C 180,E1 -27047.201,E2 -27047.201} C_VEL
LIN {X 0,Y 109.166,Z 455.37,A -85,B 0,C 180,E1 -27050.585,E2 -27050.585} C_VEL
LIN {X 0,Y 102.426,Z 458.945,A -85,B 0,C 180,E1 -27056.702,E2 -27056.702} C_VEL
LIN {X 0,Y 96.743,Z 461.252,A -85,B 0,C 180,E1 -27064.154,E2 -27064.154} C_VEL
LIN {X 0,Y 94.556,Z 461.825,A -85,B 0,C 180,E1 -27068.178,E2 -27068.178} C_VEL
LIN {X 0,Y 91.912,Z 461.787,A -85,B 0,C 180,E1 -27076.732,E2 -27076.732} C_VEL
LIN {X 0,Y 91.214,Z 460.245,A -85,B 0,C 180,E1 -27085.574,E2 -27085.574} C_VEL
LIN {X 0,Y 91.366,Z 458.832,A -85,B 0,C 180,E1 -27089.992,E2 -27089.992} C_VEL
LIN {X 0,Y 91.237,Z 455.823,A -85,B 0,C 180,E1 -27096.627,E2 -27096.627} C_VEL
LIN {X 0,Y 91.872,Z 451.707,A -85,B 0,C 180,E1 -27103.258,E2 -27103.258} C_VEL
LIN {X 0,Y 93.883,Z 445.355,A -85,B 0,C 180,E1 -27110.819,E2 -27110.819} C_VEL
LIN {X 0,Y 96.856,Z 438.429,A -85,B 0,C 180,E1 -27116.958,E2 -27116.958} C_VEL
LIN {X 0,Y 99.83,Z 431.538,A -85,B 0,C 180,E1 -27121.682,E2 -27121.682} C_VEL
LIN {X 0,Y 103.98,Z 422.78,A -85,B 0,C 180,E1 -27126.244,E2 -27126.244} C_VEL
LIN {X 0,Y 107.899,Z 413.336,A -85,B 0,C 180,E1 -27130.018,E2 -27130.018} C_VEL
LIN {X 0,Y 112.297,Z 401.609,A -85,B 0,C 180,E1 -27133.492,E2 -27133.492} C_VEL
LIN {X 0,Y 115.041,Z 393.656,A -85,B 0,C 180,E1 -27135.236,E2 -27135.236} C_VEL
LIN {X 0,Y 118.299,Z 381.649,A -85,B 0,C 180,E1 -27137.308,E2 -27137.308} C_VEL
LIN {X 0,Y 120.95,Z 369.536,A -85,B 0,C 180,E1 -27138.728,E2 -27138.728} C_VEL
LIN {X 0,Y 122.749,Z 357.12,A -85,B 0,C 180,E1 -27139.688,E2 -27139.688} C_VEL
LIN {X 0,Y 125.24,Z 325.177,A -85,B 0,C 180,E1 -27141.209,E2 -27141.209} C_VEL
LIN {X 0,Y 125.141,Z 321.37,A -85,B 0,C 180,E1 -27141.557,E2 -27141.557} C_VEL
LIN {X 0,Y 124.393,Z 317.787,A -85,B 0,C 180,E1 -27142.185,E2 -27142.185} C_VEL
LIN {X 0,Y 123.198,Z 314.443,A -85,B 0,C 180,E1 -27143.019,E2 -27143.019} C_VEL
LIN {X 0,Y 121.736,Z 311.371,A -85,B 0,C 180,E1 -27143.994,E2 -27143.994} C_VEL
LIN {X 0,Y 116.821,Z 302.293,A -85,B 0,C 180,E1 -27147.483,E2 -27147.483} C_VEL
LIN {X 0,Y 115.481,Z 299.038,A -85,B 0,C 180,E1 -27148.61,E2 -27148.61} C_VEL
LIN {X 0,Y 113.969,Z 295.789,A -85,B 0,C 180,E1 -27149.907,E2 -27149.907} C_VEL
LIN {X 0,Y 109.516,Z 288.059,A -85,B 0,C 180,E1 -27153.987,E2 -27153.987} C_VEL
LIN {X 0,Y 106.181,Z 283.148,A -85,B 0,C 180,E1 -27157.501,E2 -27157.501} C_VEL
LIN {X 0,Y 104.046,Z 279.889,A -85,B 0,C 180,E1 -27160.115,E2 -27160.115} C_VEL
LIN {X 0,Y 101.648,Z 276.451,A -85,B 0,C 180,E1 -27163.439,E2 -27163.439} C_VEL
LIN {X 0,Y 101.04,Z 275.633,A -85,B 0,C 180,E1 -27164.362,E2 -27164.362} C_VEL
LIN {X 0,Y 98.701,Z 273.007,A -85,B 0,C 180,E1 -27168.316,E2 -27168.316} C_VEL
LIN {X 0,Y 97.686,Z 270.621,A -85,B 0,C 180,E1 -27170.683,E2 -27170.683} C_VEL
LIN {X 0,Y 94.899,Z 268.169,A -85,B 0,C 180,E1 -27178.673,E2 -27178.673} C_VEL
LIN {X 0,Y 94.483,Z 267.18,A -85,B 0,C 180,E1 -27181.064,E2 -27181.064} C_VEL
LIN {X 0,Y 93.897,Z 267.181,A -85,B 0,C 180,E1 -27189.67,E2 -27189.67} C_VEL
LIN {X 0,Y 94.26,Z 268.19,A -85,B 0,C 180,E1 -27194.132,E2 -27194.132} C_VEL
LIN {X 0,Y 97.367,Z 270.773,A -85,B 0,C 180,E1 -27204.482,E2 -27204.482} C_VEL
LIN {X 0,Y 98.977,Z 273.836,A -85,B 0,C 180,E1 -27208.06,E2 -27208.06} C_VEL
LIN {X 0,Y 101.314,Z 276.142,A -85,B 0,C 180,E1 -27211.835,E2 -27211.835} C_VEL
LIN {X 0,Y 103.669,Z 279.697,A -85,B 0,C 180,E1 -27215.185,E2 -27215.185} C_VEL
LIN {X 0,Y 104.924,Z 281.301,A -85,B 0,C 180,E1 -27216.742,E2 -27216.742} C_VEL
LIN {X 0,Y 107.991,Z 285.975,A -85,B 0,C 180,E1 -27220.232,E2 -27220.232} C_VEL
LIN {X 0,Y 111.567,Z 291.521,A -85,B 0,C 180,E1 -27223.712,E2 -27223.712} C_VEL
LIN {X 0,Y 116.085,Z 299.715,A -85,B 0,C 180,E1 -27227.568,E2 -27227.568} C_VEL
LIN {X 0,Y 120.242,Z 308.712,A -85,B 0,C 180,E1 -27230.753,E2 -27230.753} C_VEL
LIN {X 0,Y 121.053,Z 310.716,A -85,B 0,C 180,E1 -27231.349,E2 -27231.349} C_VEL
LIN {X 0,Y 117.668,Z 351.31,A -85,B 0,C 180,E1 -27233.337,E2 -27233.337} C_VEL
LIN {X 0,Y 115.535,Z 364.634,A -85,B 0,C 180,E1 -27234.521,E2 -27234.521} C_VEL
LIN {X 0,Y 112.913,Z 376.659,A -85,B 0,C 180,E1 -27236.211,E2 -27236.211} C_VEL
LIN {X 0,Y 109.407,Z 388.627,A -85,B 0,C 180,E1 -27238.549,E2 -27238.549} C_VEL
LIN {X 0,Y 105.695,Z 398.83,A -85,B 0,C 180,E1 -27241.189,E2 -27241.189} C_VEL
LIN {X 0,Y 101.493,Z 409.365,A -85,B 0,C 180,E1 -27244.914,E2 -27244.914} C_VEL
LIN {X 0,Y 97.494,Z 418.023,A -85,B 0,C 180,E1 -27248.883,E2 -27248.883} C_VEL
LIN {X 0,Y 93.595,Z 425.997,A -85,B 0,C 180,E1 -27253.654,E2 -27253.654} C_VEL
LIN {X 0,Y 89.726,Z 433.782,A -85,B 0,C 180,E1 -27259.858,E2 -27259.858} C_VEL
LIN {X 0,Y 86.458,Z 440.951,A -85,B 0,C 180,E1 -27267.679,E2 -27267.679} C_VEL
LIN {X 0,Y 84.649,Z 445.844,A -85,B 0,C 180,E1 -27274.945,E2 -27274.945} C_VEL
LIN {X 0,Y 83.709,Z 449.422,A -85,B 0,C 180,E1 -27282.124,E2 -27282.124} C_VEL
LIN {X 0,Y 83.917,Z 452.062,A -85,B 0,C 180,E1 -27289.579,E2 -27289.579} C_VEL
LIN {X 0,Y 84.731,Z 453.281,A -85,B 0,C 180,E1 -27294.508,E2 -27294.508} C_VEL
LIN {X 0,Y 85.99,Z 454.056,A -85,B 0,C 180,E1 -27299.372,E2 -27299.372} C_VEL
LIN {X 0,Y 87.826,Z 454.427,A -85,B 0,C 180,E1 -27304.072,E2 -27304.072} C_VEL
LIN {X 0,Y 90.4,Z 454.361,A -85,B 0,C 180,E1 -27308.976,E2 -27308.976} C_VEL
LIN {X 0,Y 96.271,Z 452.965,A -85,B 0,C 180,E1 -27316.893,E2 -27316.893} C_VEL
LIN {X 0,Y 100.289,Z 451.514,A -85,B 0,C 180,E1 -27320.9,E2 -27320.9} C_VEL
LIN {X 0,Y 106.274,Z 448.718,A -85,B 0,C 180,E1 -27325.759,E2 -27325.759} C_VEL
LIN {X 0,Y 113.288,Z 444.693,A -85,B 0,C 180,E1 -27330.289,E2 -27330.289} C_VEL
LIN {X 0,Y 122.226,Z 438.368,A -85,B 0,C 180,E1 -27334.91,E2 -27334.91} C_VEL
LIN {X 0,Y 130.435,Z 431.39,A -85,B 0,C 180,E1 -27338.35,E2 -27338.35} C_VEL
LIN {X 0,Y 137.561,Z 424.189,A -85,B 0,C 180,E1 -27340.938,E2 -27340.938} C_VEL
LIN {X 0,Y 145.038,Z 415.376,A -85,B 0,C 180,E1 -27343.194,E2 -27343.194} C_VEL
LIN {X 0,Y 151.819,Z 405.669,A -85,B 0,C 180,E1 -27345.091,E2 -27345.091} C_VEL
LIN {X 0,Y 158.007,Z 394.941,A -85,B 0,C 180,E1 -27346.647,E2 -27346.647} C_VEL
LIN {X 0,Y 163.183,Z 383.741,A -85,B 0,C 180,E1 -27347.891,E2 -27347.891} C_VEL
LIN {X 0,Y 167.497,Z 371.578,A -85,B 0,C 180,E1 -27348.862,E2 -27348.862} C_VEL
LIN {X 0,Y 170.703,Z 358.812,A -85,B 0,C 180,E1 -27349.607,E2 -27349.607} C_VEL
LIN {X 0,Y 171.745,Z 352.86,A -85,B 0,C 180,E1 -27349.899,E2 -27349.899} C_VEL
LIN {X 0,Y 169.584,Z 347.315,A -85,B 0,C 180,E1 -27353.566,E2 -27353.566} C_VEL
LIN {X 0,Y 168.241,Z 344.317,A -85,B 0,C 180,E1 -27356.24,E2 -27356.24} C_VEL
LIN {X 0,Y 167.24,Z 341.9,A -85,B 0,C 180,E1 -27358.797,E2 -27358.797} C_VEL
LIN {X 0,Y 166.034,Z 338.442,A -85,B 0,C 180,E1 -27364.249,E2 -27364.249} C_VEL
LIN {X 0,Y 165.947,Z 338.51,A -85,B 0,C 180,E1 -27369.596,E2 -27369.596} C_VEL
LIN {X 0,Y 167.373,Z 342.69,A -85,B 0,C 180,E1 -27376.133,E2 -27376.133} C_VEL
LIN {X 0,Y 168.701,Z 346.903,A -85,B 0,C 180,E1 -27379.468,E2 -27379.468} C_VEL
LIN {X 0,Y 170.161,Z 351.907,A -85,B 0,C 180,E1 -27382.381,E2 -27382.381} C_VEL
LIN {X 0,Y 171.451,Z 357.249,A -85,B 0,C 180,E1 -27384.763,E2 -27384.763} C_VEL
LIN {X 0,Y 168.544,Z 370.847,A -85,B 0,C 180,E1 -27385.294,E2 -27385.294} C_VEL
LIN {X 0,Y 164.722,Z 382.973,A -85,B 0,C 180,E1 -27385.986,E2 -27385.986} C_VEL
LIN {X 0,Y 159.634,Z 394.941,A -85,B 0,C 180,E1 -27386.936,E2 -27386.936} C_VEL
LIN {X 0,Y 153.504,Z 406.34,A -85,B 0,C 180,E1 -27388.196,E2 -27388.196} C_VEL
LIN {X 0,Y 146.682,Z 416.65,A -85,B 0,C 180,E1 -27389.723,E2 -27389.723} C_VEL
LIN {X 0,Y 140.093,Z 425.085,A -85,B 0,C 180,E1 -27391.478,E2 -27391.478} C_VEL
LIN {X 0,Y 131.63,Z 434.256,A -85,B 0,C 180,E1 -27394.148,E2 -27394.148} C_VEL
LIN {X 0,Y 123.49,Z 441.666,A -85,B 0,C 180,E1 -27397.176,E2 -27397.176} C_VEL
LIN {X 0,Y 115.781,Z 447.648,A -85,B 0,C 180,E1 -27400.642,E2 -27400.642} C_VEL
LIN {X 0,Y 108.689,Z 452.407,A -85,B 0,C 180,E1 -27404.657,E2 -27404.657} C_VEL
LIN {X 0,Y 103.187,Z 455.604,A -85,B 0,C 180,E1 -27408.523,E2 -27408.523} C_VEL
LIN {X 0,Y 96.561,Z 458.793,A -85,B 0,C 180,E1 -27414.385,E2 -27414.385} C_VEL
LIN {X 0,Y 90.376,Z 461.016,A -85,B 0,C 180,E1 -27422.181,E2 -27422.181} C_VEL
LIN {X 0,Y 86.222,Z 461.644,A -85,B 0,C 180,E1 -27430.965,E2 -27430.965} C_VEL
LIN {X 0,Y 84.309,Z 460.781,A -85,B 0,C 180,E1 -27440.395,E2 -27440.395} C_VEL
LIN {X 0,Y 84.138,Z 459.76,A -85,B 0,C 180,E1 -27445.201,E2 -27445.201} C_VEL
LIN {X 0,Y 84.278,Z 458.291,A -85,B 0,C 180,E1 -27449.992,E2 -27449.992} C_VEL
LIN {X 0,Y 84.159,Z 455.195,A -85,B 0,C 180,E1 -27457.187,E2 -27457.187} C_VEL
LIN {X 0,Y 84.935,Z 450.989,A -85,B 0,C 180,E1 -27464.363,E2 -27464.363} C_VEL
LIN {X 0,Y 87.259,Z 444.54,A -85,B 0,C 180,E1 -27472.482,E2 -27472.482} C_VEL
LIN {X 0,Y 90.508,Z 437.485,A -85,B 0,C 180,E1 -27479.021,E2 -27479.021} C_VEL
LIN {X 0,Y 94.398,Z 429.16,A -85,B 0,C 180,E1 -27484.772,E2 -27484.772} C_VEL
LIN {X 0,Y 98.282,Z 421.5,A -85,B 0,C 180,E1 -27488.719,E2 -27488.719} C_VEL
LIN {X 0,Y 102.543,Z 411.861,A -85,B 0,C 180,E1 -27492.58,E2 -27492.58} C_VEL
LIN {X 0,Y 106.672,Z 401.324,A -85,B 0,C 180,E1 -27495.751,E2 -27495.751} C_VEL
LIN {X 0,Y 109.546,Z 393.377,A -85,B 0,C 180,E1 -27497.528,E2 -27497.528} C_VEL
LIN {X 0,Y 113.309,Z 380.266,A -85,B 0,C 180,E1 -27499.774,E2 -27499.774} C_VEL
LIN {X 0,Y 116.04,Z 367.617,A -85,B 0,C 180,E1 -27501.224,E2 -27501.224} C_VEL
LIN {X 0,Y 117.79,Z 354.858,A -85,B 0,C 180,E1 -27502.159,E2 -27502.159} C_VEL
LIN {X 0,Y 120.342,Z 322.308,A -85,B 0,C 180,E1 -27503.75,E2 -27503.75} C_VEL
LIN {X 0,Y 119.955,Z 312.932,A -85,B 0,C 180,E1 -27504.768,E2 -27504.768} C_VEL
LIN {X 0,Y 117.126,Z 303.621,A -85,B 0,C 180,E1 -27507.177,E2 -27507.177} C_VEL
LIN {X 0,Y 115.481,Z 299.038,A -85,B 0,C 180,E1 -27508.61,E2 -27508.61} C_VEL
LIN {X 0,Y 114.128,Z 296.212,A -85,B 0,C 180,E1 -27509.76,E2 -27509.76} C_VEL
LIN {X 0,Y 112.439,Z 293.984,A -85,B 0,C 180,E1 -27511.142,E2 -27511.142} C_VEL
LIN {X 0,Y 109.607,Z 291.515,A -85,B 0,C 180,E1 -27513.523,E2 -27513.523} C_VEL
LIN {X 0,Y 103.068,Z 287.301,A -85,B 0,C 180,E1 -27520.058,E2 -27520.058} C_VEL
LIN {X 0,Y 101.534,Z 285.753,A -85,B 0,C 180,E1 -27522.021,E2 -27522.021} C_VEL
LIN {X 0,Y 99.199,Z 282.154,A -85,B 0,C 180,E1 -27525.674,E2 -27525.674} C_VEL
LIN {X 0,Y 96.901,Z 279.226,A -85,B 0,C 180,E1 -27530.03,E2 -27530.03} C_VEL
LIN {X 0,Y 96.102,Z 277.317,A -85,B 0,C 180,E1 -27532.117,E2 -27532.117} C_VEL
LIN {X 0,Y 93.776,Z 274.962,A -85,B 0,C 180,E1 -27539.73,E2 -27539.73} C_VEL
LIN {X 0,Y 93.408,Z 274.171,A -85,B 0,C 180,E1 -27542.155,E2 -27542.155} C_VEL
LIN {X 0,Y 93.018,Z 274.269,A -85,B 0,C 180,E1 -27549.889,E2 -27549.889} C_VEL
LIN {X 0,Y 95.959,Z 277.717,A -85,B 0,C 180,E1 -27563.43,E2 -27563.43} C_VEL
LIN {X 0,Y 97.743,Z 280.857,A -85,B 0,C 180,E1 -27567.571,E2 -27567.571} C_VEL
LIN {X 0,Y 99.418,Z 282.69,A -85,B 0,C 180,E1 -27570.487,E2 -27570.487} C_VEL
LIN {X 0,Y 101.84,Z 286.314,A -85,B 0,C 180,E1 -27574.177,E2 -27574.177} C_VEL
LIN {X 0,Y 105.169,Z 291.554,A -85,B 0,C 180,E1 -27578.422,E2 -27578.422} C_VEL
LIN {X 0,Y 108.592,Z 297.193,A -85,B 0,C 180,E1 -27582.104,E2 -27582.104} C_VEL
LIN {X 0,Y 112.664,Z 305.109,A -85,B 0,C 180,E1 -27585.941,E2 -27585.941} C_VEL
LIN {X 0,Y 116.168,Z 313.174,A -85,B 0,C 180,E1 -27588.917,E2 -27588.917} C_VEL
LIN {X 0,Y 112.824,Z 351.124,A -85,B 0,C 180,E1 -27590.761,E2 -27590.761} C_VEL
LIN {X 0,Y 110.52,Z 364.955,A -85,B 0,C 180,E1 -27591.985,E2 -27591.985} C_VEL
LIN {X 0,Y 107.663,Z 377.297,A -85,B 0,C 180,E1 -27593.743,E2 -27593.743} C_VEL
LIN {X 0,Y 103.96,Z 389.186,A -85,B 0,C 180,E1 -27596.113,E2 -27596.113} C_VEL
LIN {X 0,Y 100.045,Z 399.345,A -85,B 0,C 180,E1 -27598.808,E2 -27598.808} C_VEL
LIN {X 0,Y 95.579,Z 409.847,A -85,B 0,C 180,E1 -27602.652,E2 -27602.652} C_VEL
LIN {X 0,Y 90.863,Z 419.359,A -85,B 0,C 180,E1 -27607.259,E2 -27607.259} C_VEL
LIN {X 0,Y 85.987,Z 428.513,A -85,B 0,C 180,E1 -27613.387,E2 -27613.387} C_VEL
LIN {X 0,Y 82.083,Z 435.893,A -85,B 0,C 180,E1 -27620.15,E2 -27620.15} C_VEL
LIN {X 0,Y 79.281,Z 441.803,A -85,B 0,C 180,E1 -27627.469,E2 -27627.469} C_VEL
LIN {X 0,Y 77.434,Z 446.476,A -85,B 0,C 180,E1 -27635.216,E2 -27635.216} C_VEL
LIN {X 0,Y 76.572,Z 450.059,A -85,B 0,C 180,E1 -27643.273,E2 -27643.273} C_VEL
LIN {X 0,Y 77.012,Z 452.609,A -85,B 0,C 180,E1 -27651.417,E2 -27651.417} C_VEL
LIN {X 0,Y 78.054,Z 453.741,A -85,B 0,C 180,E1 -27656.764,E2 -27656.764} C_VEL
LIN {X 0,Y 79.601,Z 454.469,A -85,B 0,C 180,E1 -27661.995,E2 -27661.995} C_VEL
LIN {X 0,Y 81.77,Z 454.793,A -85,B 0,C 180,E1 -27666.994,E2 -27666.994} C_VEL
LIN {X 0,Y 84.472,Z 454.67,A -85,B 0,C 180,E1 -27671.734,E2 -27671.734} C_VEL
LIN {X 0,Y 87.669,Z 454.11,A -85,B 0,C 180,E1 -27676.183,E2 -27676.183} C_VEL
LIN {X 0,Y 94.959,Z 451.911,A -85,B 0,C 180,E1 -27683.696,E2 -27683.696} C_VEL
LIN {X 0,Y 102.262,Z 448.716,A -85,B 0,C 180,E1 -27689.217,E2 -27689.217} C_VEL
LIN {X 0,Y 109.782,Z 444.563,A -85,B 0,C 180,E1 -27693.673,E2 -27693.673} C_VEL
LIN {X 0,Y 119.253,Z 438.103,A -85,B 0,C 180,E1 -27698.159,E2 -27698.159} C_VEL
LIN {X 0,Y 127.876,Z 430.979,A -85,B 0,C 180,E1 -27701.453,E2 -27701.453} C_VEL
LIN {X 0,Y 135.326,Z 423.605,A -85,B 0,C 180,E1 -27703.899,E2 -27703.899} C_VEL
LIN {X 0,Y 143.593,Z 413.862,A -85,B 0,C 180,E1 -27706.182,E2 -27706.182} C_VEL
LIN {X 0,Y 150.885,Z 403.389,A -85,B 0,C 180,E1 -27707.997,E2 -27707.997} C_VEL
LIN {X 0,Y 157.259,Z 391.913,A -85,B 0,C 180,E1 -27709.477,E2 -27709.477} C_VEL
LIN {X 0,Y 162.461,Z 380.03,A -85,B 0,C 180,E1 -27710.606,E2 -27710.606} C_VEL
LIN {X 0,Y 166.644,Z 367.338,A -85,B 0,C 180,E1 -27711.457,E2 -27711.457} C_VEL
LIN {X 0,Y 168.99,Z 357.071,A -85,B 0,C 180,E1 -27712.031,E2 -27712.031} C_VEL
LIN {X 0,Y 167.323,Z 351.899,A -85,B 0,C 180,E1 -27715.936,E2 -27715.936} C_VEL
LIN {X 0,Y 166.089,Z 348.693,A -85,B 0,C 180,E1 -27719.395,E2 -27719.395} C_VEL
LIN {X 0,Y 165.072,Z 345.387,A -85,B 0,C 180,E1 -27724.885,E2 -27724.885} C_VEL
LIN {X 0,Y 165.027,Z 345.465,A -85,B 0,C 180,E1 -27729.19,E2 -27729.19} C_VEL
LIN {X 0,Y 166.176,Z 349.291,A -85,B 0,C 180,E1 -27735.328,E2 -27735.328} C_VEL
LIN {X 0,Y 167.215,Z 353.315,A -85,B 0,C 180,E1 -27738.534,E2 -27738.534} C_VEL
LIN {X 0,Y 168.218,Z 357.784,A -85,B 0,C 180,E1 -27741.202,E2 -27741.202} C_VEL
LIN {X 0,Y 168.73,Z 360.483,A -85,B 0,C 180,E1 -27742.527,E2 -27742.527} C_VEL
LIN {X 0,Y 166.028,Z 372.039,A -85,B 0,C 180,E1 -27743.031,E2 -27743.031} C_VEL
LIN {X 0,Y 161.846,Z 384.392,A -85,B 0,C 180,E1 -27743.733,E2 -27743.733} C_VEL
LIN {X 0,Y 156.571,Z 396.139,A -85,B 0,C 180,E1 -27744.639,E2 -27744.639} C_VEL
LIN {X 0,Y 150.3,Z 407.26,A -85,B 0,C 180,E1 -27745.826,E2 -27745.826} C_VEL
LIN {X 0,Y 142.554,Z 418.277,A -85,B 0,C 180,E1 -27747.45,E2 -27747.45} C_VEL
LIN {X 0,Y 135.091,Z 427.193,A -85,B 0,C 180,E1 -27749.377,E2 -27749.377} C_VEL
LIN {X 0,Y 127.788,Z 434.585,A -85,B 0,C 180,E1 -27751.518,E2 -27751.518} C_VEL
LIN {X 0,Y 119.335,Z 441.881,A -85,B 0,C 180,E1 -27754.459,E2 -27754.459} C_VEL
LIN {X 0,Y 111.288,Z 447.76,A -85,B 0,C 180,E1 -27757.868,E2 -27757.868} C_VEL
LIN {X 0,Y 103.799,Z 452.426,A -85,B 0,C 180,E1 -27761.855,E2 -27761.855} C_VEL
LIN {X 0,Y 97.349,Z 455.838,A -85,B 0,C 180,E1 -27766.217,E2 -27766.217} C_VEL
LIN {X 0,Y 90.876,Z 458.642,A -85,B 0,C 180,E1 -27771.774,E2 -27771.774} C_VEL
LIN {X 0,Y 87.254,Z 459.905,A -85,B 0,C 180,E1 -27775.673,E2 -27775.673} C_VEL
LIN {X 0,Y 81.488,Z 461.207,A -85,B 0,C 180,E1 -27784.447,E2 -27784.447} C_VEL
LIN {X 0,Y 78.114,Z 461.012,A -85,B 0,C 180,E1 -27794.333,E2 -27794.333} C_VEL
LIN {X 0,Y 77.303,Z 460.348,A -85,B 0,C 180,E1 -27799.515,E2 -27799.515} C_VEL
LIN {X 0,Y 77.056,Z 459.255,A -85,B 0,C 180,E1 -27804.758,E2 -27804.758} C_VEL
LIN {X 0,Y 77.192,Z 457.747,A -85,B 0,C 180,E1 -27809.991,E2 -27809.991} C_VEL
LIN {X 0,Y 77.108,Z 454.564,A -85,B 0,C 180,E1 -27817.848,E2 -27817.848} C_VEL
LIN {X 0,Y 78.02,Z 450.263,A -85,B 0,C 180,E1 -27825.668,E2 -27825.668} C_VEL
LIN {X 0,Y 80.718,Z 443.719,A -85,B 0,C 180,E1 -27834.418,E2 -27834.418} C_VEL
LIN {X 0,Y 84.3,Z 436.492,A -85,B 0,C 180,E1 -27841.39,E2 -27841.39} C_VEL
LIN {X 0,Y 88.124,Z 428.953,A -85,B 0,C 180,E1 -27846.855,E2 -27846.855} C_VEL
LIN {X 0,Y 91.84,Z 422.179,A -85,B 0,C 180,E1 -27850.562,E2 -27850.562} C_VEL
LIN {X 0,Y 96.311,Z 412.753,A -85,B 0,C 180,E1 -27854.601,E2 -27854.601} C_VEL
LIN {X 0,Y 100.675,Z 402.486,A -85,B 0,C 180,E1 -27857.862,E2 -27857.862} C_VEL
LIN {X 0,Y 104.247,Z 393.1,A -85,B 0,C 180,E1 -27860.057,E2 -27860.057} C_VEL
LIN {X 0,Y 108.203,Z 380.003,A -85,B 0,C 180,E1 -27862.318,E2 -27862.318} C_VEL
LIN {X 0,Y 111.055,Z 367.386,A -85,B 0,C 180,E1 -27863.773,E2 -27863.773} C_VEL
LIN {X 0,Y 112.963,Z 353.953,A -85,B 0,C 180,E1 -27864.748,E2 -27864.748} C_VEL
LIN {X 0,Y 115.51,Z 322.963,A -85,B 0,C 180,E1 -27866.275,E2 -27866.275} C_VEL
LIN {X 0,Y 115.297,Z 315.419,A -85,B 0,C 180,E1 -27867.119,E2 -27867.119} C_VEL
LIN {X 0,Y 112.756,Z 306.695,A -85,B 0,C 180,E1 -27869.573,E2 -27869.573} C_VEL
LIN {X 0,Y 110.87,Z 301.47,A -85,B 0,C 180,E1 -27871.426,E2 -27871.426} C_VEL
LIN {X 0,Y 106.55,Z 293.597,A -85,B 0,C 180,E1 -27875.782,E2 -27875.782} C_VEL
LIN {X 0,Y 102.143,Z 286.437,A -85,B 0,C 180,E1 -27881.211,E2 -27881.211} C_VEL
LIN {X 0,Y 101.534,Z 285.753,A -85,B 0,C 180,E1 -27882.021,E2 -27882.021} C_VEL
LIN {X 0,Y 100.099,Z 284.563,A -85,B 0,C 180,E1 -27883.999,E2 -27883.999} C_VEL
LIN {X 0,Y 97.683,Z 284.105,A -85,B 0,C 180,E1 -27887.571,E2 -27887.571} C_VEL
LIN {X 0,Y 95.176,Z 284.229,A -85,B 0,C 180,E1 -27892.178,E2 -27892.178} C_VEL
LIN {X 0,Y 94.519,Z 284.001,A -85,B 0,C 180,E1 -27893.759,E2 -27893.759} C_VEL
LIN {X 0,Y 92.617,Z 281.523,A -85,B 0,C 180,E1 -27901.357,E2 -27901.357} C_VEL
LIN {X 0,Y 92.259,Z 281.123,A -85,B 0,C 180,E1 -27904.367,E2 -27904.367} C_VEL
LIN {X 0,Y 92.165,Z 281.424,A -85,B 0,C 180,E1 -27910.588,E2 -27910.588} C_VEL
LIN {X 0,Y 94.588,Z 284.612,A -85,B 0,C 180,E1 -27922.338,E2 -27922.338} C_VEL
LIN {X 0,Y 96.517,Z 287.874,A -85,B 0,C 180,E1 -27927.07,E2 -27927.07} C_VEL
LIN {X 0,Y 97.649,Z 289.319,A -85,B 0,C 180,E1 -27929.212,E2 -27929.212} C_VEL
LIN {X 0,Y 100.657,Z 294.134,A -85,B 0,C 180,E1 -27934.068,E2 -27934.068} C_VEL
LIN {X 0,Y 104.163,Z 300.008,A -85,B 0,C 180,E1 -27938.625,E2 -27938.625} C_VEL
LIN {X 0,Y 108.129,Z 307.758,A -85,B 0,C 180,E1 -27942.989,E2 -27942.989} C_VEL
LIN {X 0,Y 111.478,Z 315.53,A -85,B 0,C 180,E1 -27946.245,E2 -27946.245} C_VEL
LIN {X 0,Y 108.156,Z 351.489,A -85,B 0,C 180,E1 -27948.002,E2 -27948.002} C_VEL
LIN {X 0,Y 105.796,Z 364.972,A -85,B 0,C 180,E1 -27949.176,E2 -27949.176} C_VEL
LIN {X 0,Y 102.634,Z 377.924,A -85,B 0,C 180,E1 -27951.027,E2 -27951.027} C_VEL
LIN {X 0,Y 98.715,Z 389.748,A -85,B 0,C 180,E1 -27953.41,E2 -27953.41} C_VEL
LIN {X 0,Y 94.589,Z 399.861,A -85,B 0,C 180,E1 -27956.146,E2 -27956.146} C_VEL
LIN {X 0,Y 89.834,Z 410.328,A -85,B 0,C 180,E1 -27960.096,E2 -27960.096} C_VEL
LIN {X 0,Y 84.967,Z 419.512,A -85,B 0,C 180,E1 -27964.702,E2 -27964.702} C_VEL
LIN {X 0,Y 79.969,Z 428.25,A -85,B 0,C 180,E1 -27970.769,E2 -27970.769} C_VEL
LIN {X 0,Y 75.645,Z 435.735,A -85,B 0,C 180,E1 -27977.944,E2 -27977.944} C_VEL
LIN {X 0,Y 72.952,Z 440.817,A -85,B 0,C 180,E1 -27984.482,E2 -27984.482} C_VEL
LIN {X 0,Y 70.887,Z 445.363,A -85,B 0,C 180,E1 -27992.067,E2 -27992.067} C_VEL
LIN {X 0,Y 69.521,Z 449.612,A -85,B 0,C 180,E1 -28001.674,E2 -28001.674} C_VEL
LIN {X 0,Y 69.52,Z 451.605,A -85,B 0,C 180,E1 -28007.663,E2 -28007.663} C_VEL
LIN {X 0,Y 70.869,Z 453.779,A -85,B 0,C 180,E1 -28016.812,E2 -28016.812} C_VEL
LIN {X 0,Y 73.414,Z 454.883,A -85,B 0,C 180,E1 -28025.065,E2 -28025.065} C_VEL
LIN {X 0,Y 78.161,Z 455.055,A -85,B 0,C 180,E1 -28034.003,E2 -28034.003} C_VEL
LIN {X 0,Y 82.68,Z 454.332,A -85,B 0,C 180,E1 -28039.916,E2 -28039.916} C_VEL
LIN {X 0,Y 90.019,Z 452.27,A -85,B 0,C 180,E1 -28046.874,E2 -28046.874} C_VEL
LIN {X 0,Y 98.655,Z 448.684,A -85,B 0,C 180,E1 -28052.938,E2 -28052.938} C_VEL
LIN {X 0,Y 106.687,Z 444.419,A -85,B 0,C 180,E1 -28057.261,E2 -28057.261} C_VEL
LIN {X 0,Y 115.228,Z 438.874,A -85,B 0,C 180,E1 -28060.978,E2 -28060.978} C_VEL
LIN {X 0,Y 124.183,Z 431.861,A -85,B 0,C 180,E1 -28064.176,E2 -28064.176} C_VEL
LIN {X 0,Y 131.896,Z 424.626,A -85,B 0,C 180,E1 -28066.518,E2 -28066.518} C_VEL
LIN {X 0,Y 140.483,Z 414.968,A -85,B 0,C 180,E1 -28068.718,E2 -28068.718} C_VEL
LIN {X 0,Y 147.888,Z 404.791,A -85,B 0,C 180,E1 -28070.43,E2 -28070.43} C_VEL
LIN {X 0,Y 154.432,Z 393.716,A -85,B 0,C 180,E1 -28071.809,E2 -28071.809} C_VEL
LIN {X 0,Y 159.874,Z 381.938,A -85,B 0,C 180,E1 -28072.906,E2 -28072.906} C_VEL
LIN {X 0,Y 164.378,Z 369.122,A -85,B 0,C 180,E1 -28073.734,E2 -28073.734} C_VEL
LIN {X 0,Y 166.318,Z 361.57,A -85,B 0,C 180,E1 -28074.163,E2 -28074.163} C_VEL
LIN {X 0,Y 165.402,Z 357.935,A -85,B 0,C 180,E1 -28077.261,E2 -28077.261} C_VEL
LIN {X 0,Y 164.705,Z 355.462,A -85,B 0,C 180,E1 -28080.001,E2 -28080.001} C_VEL
LIN {X 0,Y 164.084,Z 352.409,A -85,B 0,C 180,E1 -28084.915,E2 -28084.915} C_VEL
LIN {X 0,Y 164.02,Z 352.52,A -85,B 0,C 180,E1 -28088.909,E2 -28088.909} C_VEL
LIN {X 0,Y 164.857,Z 356.208,A -85,B 0,C 180,E1 -28094.821,E2 -28094.821} C_VEL
LIN {X 0,Y 165.469,Z 359.427,A -85,B 0,C 180,E1 -28097.456,E2 -28097.456} C_VEL
LIN {X 0,Y 166.064,Z 363.633,A -85,B 0,C 180,E1 -28100.018,E2 -28100.018} C_VEL
LIN {X 0,Y 166.114,Z 364.426,A -85,B 0,C 180,E1 -28100.372,E2 -28100.372} C_VEL
LIN {X 0,Y 162.645,Z 376.825,A -85,B 0,C 180,E1 -28100.902,E2 -28100.902} C_VEL
LIN {X 0,Y 157.81,Z 389.133,A -85,B 0,C 180,E1 -28101.62,E2 -28101.62} C_VEL
LIN {X 0,Y 151.366,Z 401.679,A -85,B 0,C 180,E1 -28102.661,E2 -28102.661} C_VEL
LIN {X 0,Y 144.196,Z 412.736,A -85,B 0,C 180,E1 -28103.955,E2 -28103.955} C_VEL
LIN {X 0,Y 137.919,Z 420.816,A -85,B 0,C 180,E1 -28105.245,E2 -28105.245} C_VEL
LIN {X 0,Y 130.235,Z 429.224,A -85,B 0,C 180,E1 -28107.074,E2 -28107.074} C_VEL
LIN {X 0,Y 122.771,Z 436.23,A -85,B 0,C 180,E1 -28109.19,E2 -28109.19} C_VEL
LIN {X 0,Y 114.056,Z 443.12,A -85,B 0,C 180,E1 -28112.082,E2 -28112.082} C_VEL
LIN {X 0,Y 104.382,Z 449.486,A -85,B 0,C 180,E1 -28116.099,E2 -28116.099} C_VEL
LIN {X 0,Y 96.719,Z 453.694,A -85,B 0,C 180,E1 -28120.268,E2 -28120.268} C_VEL
LIN {X 0,Y 89.677,Z 456.878,A -85,B 0,C 180,E1 -28125.138,E2 -28125.138} C_VEL
LIN {X 0,Y 85.406,Z 458.49,A -85,B 0,C 180,E1 -28128.822,E2 -28128.822} C_VEL
LIN {X 0,Y 81.464,Z 459.695,A -85,B 0,C 180,E1 -28132.844,E2 -28132.844} C_VEL
LIN {X 0,Y 75.117,Z 460.898,A -85,B 0,C 180,E1 -28142.101,E2 -28142.101} C_VEL
LIN {X 0,Y 71.295,Z 460.625,A -85,B 0,C 180,E1 -28152.79,E2 -28152.79} C_VEL
LIN {X 0,Y 70.004,Z 458.752,A -85,B 0,C 180,E1 -28164.229,E2 -28164.229} C_VEL
LIN {X 0,Y 70.091,Z 457.202,A -85,B 0,C 180,E1 -28169.99,E2 -28169.99} C_VEL
LIN {X 0,Y 70.049,Z 453.931,A -85,B 0,C 180,E1 -28178.645,E2 -28178.645} C_VEL
LIN {X 0,Y 71.167,Z 449.538,A -85,B 0,C 180,E1 -28187.221,E2 -28187.221} C_VEL
LIN {X 0,Y 73.695,Z 443.918,A -85,B 0,C 180,E1 -28195.4,E2 -28195.4} C_VEL
LIN {X 0,Y 77.517,Z 436.867,A -85,B 0,C 180,E1 -28202.941,E2 -28202.941} C_VEL
LIN {X 0,Y 81.984,Z 428.744,A -85,B 0,C 180,E1 -28209.253,E2 -28209.253} C_VEL
LIN {X 0,Y 86.515,Z 420.899,A -85,B 0,C 180,E1 -28213.653,E2 -28213.653} C_VEL
LIN {X 0,Y 91.373,Z 411.278,A -85,B 0,C 180,E1 -28217.741,E2 -28217.741} C_VEL
LIN {X 0,Y 96.006,Z 400.753,A -85,B 0,C 180,E1 -28221.04,E2 -28221.04} C_VEL
LIN {X 0,Y 99.174,Z 392.823,A -85,B 0,C 180,E1 -28222.849,E2 -28222.849} C_VEL
LIN {X 0,Y 103.319,Z 379.779,A -85,B 0,C 180,E1 -28225.103,E2 -28225.103} C_VEL
LIN {X 0,Y 106.202,Z 367.768,A -85,B 0,C 180,E1 -28226.497,E2 -28226.497} C_VEL
LIN {X 0,Y 108.153,Z 355.364,A -85,B 0,C 180,E1 -28227.428,E2 -28227.428} C_VEL
LIN {X 0,Y 110.932,Z 323.52,A -85,B 0,C 180,E1 -28229.018,E2 -28229.018} C_VEL
LIN {X 0,Y 110.805,Z 317.627,A -85,B 0,C 180,E1 -28229.723,E2 -28229.723} C_VEL
LIN {X 0,Y 108.338,Z 308.923,A -85,B 0,C 180,E1 -28232.452,E2 -28232.452} C_VEL
LIN {X 0,Y 106.993,Z 305.464,A -85,B 0,C 180,E1 -28233.922,E2 -28233.922} C_VEL
LIN {X 0,Y 103.573,Z 298.948,A -85,B 0,C 180,E1 -28237.823,E2 -28237.823} C_VEL
LIN {X 0,Y 99.854,Z 292.533,A -85,B 0,C 180,E1 -28242.919,E2 -28242.919} C_VEL
LIN {X 0,Y 97.325,Z 288.598,A -85,B 0,C 180,E1 -28247.189,E2 -28247.189} C_VEL
LIN {X 0,Y 95.156,Z 285.359,A -85,B 0,C 180,E1 -28251.905,E2 -28251.905} C_VEL
LIN {X 0,Y 94.519,Z 284.001,A -85,B 0,C 180,E1 -28253.759,E2 -28253.759} C_VEL
LIN {X 0,Y 93.294,Z 283.821,A -85,B 0,C 180,E1 -28257.302,E2 -28257.302} C_VEL
LIN {X 0,Y 92.318,Z 284.598,A -85,B 0,C 180,E1 -28260.903,E2 -28260.903} C_VEL
LIN {X 0,Y 91.448,Z 289.289,A -85,B 0,C 180,E1 -28273.137,E2 -28273.137} C_VEL
LIN {X 0,Y 93.274,Z 291.462,A -85,B 0,C 180,E1 -28281.259,E2 -28281.259} C_VEL
LIN {X 0,Y 95.045,Z 294.593,A -85,B 0,C 180,E1 -28286.019,E2 -28286.019} C_VEL
LIN {X 0,Y 95.855,Z 295.743,A -85,B 0,C 180,E1 -28287.716,E2 -28287.716} C_VEL
LIN {X 0,Y 98.586,Z 300.478,A -85,B 0,C 180,E1 -28292.612,E2 -28292.612} C_VEL
LIN {X 0,Y 102.012,Z 306.781,A -85,B 0,C 180,E1 -28297.471,E2 -28297.471} C_VEL
LIN {X 0,Y 105.166,Z 313.534,A -85,B 0,C 180,E1 -28301.297,E2 -28301.297} C_VEL
LIN {X 0,Y 107.103,Z 318.271,A -85,B 0,C 180,E1 -28303.43,E2 -28303.43} C_VEL
LIN {X 0,Y 103.7,Z 352.189,A -85,B 0,C 180,E1 -28305.018,E2 -28305.018} C_VEL
LIN {X 0,Y 101.212,Z 365.728,A -85,B 0,C 180,E1 -28306.209,E2 -28306.209} C_VEL
LIN {X 0,Y 97.859,Z 378.541,A -85,B 0,C 180,E1 -28308.04,E2 -28308.04} C_VEL
LIN {X 0,Y 93.713,Z 390.31,A -85,B 0,C 180,E1 -28310.411,E2 -28310.411} C_VEL
LIN {X 0,Y 89.361,Z 400.377,A -85,B 0,C 180,E1 -28313.167,E2 -28313.167} C_VEL
LIN {X 0,Y 84.327,Z 410.713,A -85,B 0,C 180,E1 -28317.145,E2 -28317.145} C_VEL
LIN {X 0,Y 79.013,Z 420.083,A -85,B 0,C 180,E1 -28322.031,E2 -28322.031} C_VEL
LIN {X 0,Y 73.244,Z 429.364,A -85,B 0,C 180,E1 -28328.923,E2 -28328.923} C_VEL
LIN {X 0,Y 68.666,Z 436.71,A -85,B 0,C 180,E1 -28336.698,E2 -28336.698} C_VEL
LIN {X 0,Y 65.801,Z 441.673,A -85,B 0,C 180,E1 -28343.88,E2 -28343.88} C_VEL
LIN {X 0,Y 63.382,Z 446.755,A -85,B 0,C 180,E1 -28353.695,E2 -28353.695} C_VEL
LIN {X 0,Y 62.366,Z 450.264,A -85,B 0,C 180,E1 -28363.036,E2 -28363.036} C_VEL
LIN {X 0,Y 62.576,Z 452.184,A -85,B 0,C 180,E1 -28369.7,E2 -28369.7} C_VEL
LIN {X 0,Y 64.084,Z 454.077,A -85,B 0,C 180,E1 -28378.68,E2 -28378.68} C_VEL
LIN {X 0,Y 67.462,Z 455.294,A -85,B 0,C 180,E1 -28388.696,E2 -28388.696} C_VEL
LIN {X 0,Y 72.329,Z 455.398,A -85,B 0,C 180,E1 -28397.146,E2 -28397.146} C_VEL
LIN {X 0,Y 78.092,Z 454.554,A -85,B 0,C 180,E1 -28404.1,E2 -28404.1} C_VEL
LIN {X 0,Y 85.256,Z 452.66,A -85,B 0,C 180,E1 -28410.358,E2 -28410.358} C_VEL
LIN {X 0,Y 92.765,Z 449.863,A -85,B 0,C 180,E1 -28415.393,E2 -28415.393} C_VEL
LIN {X 0,Y 100.821,Z 446.05,A -85,B 0,C 180,E1 -28419.603,E2 -28419.603} C_VEL
LIN {X 0,Y 109.99,Z 440.689,A -85,B 0,C 180,E1 -28423.43,E2 -28423.43} C_VEL
LIN {X 0,Y 119.762,Z 433.587,A -85,B 0,C 180,E1 -28426.746,E2 -28426.746} C_VEL
LIN {X 0,Y 128.755,Z 425.654,A -85,B 0,C 180,E1 -28429.272,E2 -28429.272} C_VEL
LIN {X 0,Y 137.524,Z 416.285,A -85,B 0,C 180,E1 -28431.327,E2 -28431.327} C_VEL
LIN {X 0,Y 145.171,Z 406.228,A -85,B 0,C 180,E1 -28432.947,E2 -28432.947} C_VEL
LIN {X 0,Y 152.399,Z 394.487,A -85,B 0,C 180,E1 -28434.33,E2 -28434.33} C_VEL
LIN {X 0,Y 157.674,Z 383.561,A -85,B 0,C 180,E1 -28435.297,E2 -28435.297} C_VEL
LIN {X 0,Y 162.42,Z 370.691,A -85,B 0,C 180,E1 -28436.081,E2 -28436.081} C_VEL
LIN {X 0,Y 163.721,Z 366.154,A -85,B 0,C 180,E1 -28436.342,E2 -28436.342} C_VEL
LIN {X 0,Y 163.155,Z 362.808,A -85,B 0,C 180,E1 -28439.692,E2 -28439.692} C_VEL
LIN {X 0,Y 162.699,Z 359.371,A -85,B 0,C 180,E1 -28445.306,E2 -28445.306} C_VEL
LIN {X 0,Y 162.676,Z 359.6,A -85,B 0,C 180,E1 -28448.822,E2 -28448.822} C_VEL
LIN {X 0,Y 163.161,Z 362.9,A -85,B 0,C 180,E1 -28454.182,E2 -28454.182} C_VEL
LIN {X 0,Y 163.506,Z 365.99,A -85,B 0,C 180,E1 -28456.706,E2 -28456.706} C_VEL
LIN {X 0,Y 163.65,Z 367.96,A -85,B 0,C 180,E1 -28458.028,E2 -28458.028} C_VEL
LIN {X 0,Y 160.188,Z 379.073,A -85,B 0,C 180,E1 -28458.556,E2 -28458.556} C_VEL
LIN {X 0,Y 155.357,Z 390.609,A -85,B 0,C 180,E1 -28459.208,E2 -28459.208} C_VEL
LIN {X 0,Y 149.616,Z 401.392,A -85,B 0,C 180,E1 -28460.037,E2 -28460.037} C_VEL
LIN {X 0,Y 142.288,Z 412.44,A -85,B 0,C 180,E1 -28461.205,E2 -28461.205} C_VEL
LIN {X 0,Y 135.06,Z 421.407,A -85,B 0,C 180,E1 -28462.534,E2 -28462.534} C_VEL
LIN {X 0,Y 127.175,Z 429.653,A -85,B 0,C 180,E1 -28464.239,E2 -28464.239} C_VEL
LIN {X 0,Y 119.469,Z 436.521,A -85,B 0,C 180,E1 -28466.217,E2 -28466.217} C_VEL
LIN {X 0,Y 110.447,Z 443.291,A -85,B 0,C 180,E1 -28468.958,E2 -28468.958} C_VEL
LIN {X 0,Y 100.369,Z 449.55,A -85,B 0,C 180,E1 -28472.828,E2 -28472.828} C_VEL
LIN {X 0,Y 92.268,Z 453.668,A -85,B 0,C 180,E1 -28476.886,E2 -28476.886} C_VEL
LIN {X 0,Y 84.772,Z 456.767,A -85,B 0,C 180,E1 -28481.736,E2 -28481.736} C_VEL
LIN {X 0,Y 80.179,Z 458.334,A -85,B 0,C 180,E1 -28485.467,E2 -28485.467} C_VEL
LIN {X 0,Y 72.164,Z 460.214,A -85,B 0,C 180,E1 -28494.236,E2 -28494.236} C_VEL
LIN {X 0,Y 66.375,Z 460.599,A -85,B 0,C 180,E1 -28504.933,E2 -28504.933} C_VEL
LIN {X 0,Y 64.515,Z 460.216,A -85,B 0,C 180,E1 -28510.915,E2 -28510.915} C_VEL
LIN {X 0,Y 62.947,Z 458.248,A -85,B 0,C 180,E1 -28523.579,E2 -28523.579} C_VEL
LIN {X 0,Y 63.002,Z 456.658,A -85,B 0,C 180,E1 -28529.989,E2 -28529.989} C_VEL
LIN {X 0,Y 63.028,Z 453.301,A -85,B 0,C 180,E1 -28539.616,E2 -28539.616} C_VEL
LIN {X 0,Y 64.383,Z 448.815,A -85,B 0,C 180,E1 -28549.102,E2 -28549.102} C_VEL
LIN {X 0,Y 67.333,Z 443.097,A -85,B 0,C 180,E1 -28558,E2 -28558} C_VEL
LIN {X 0,Y 71.607,Z 435.877,A -85,B 0,C 180,E1 -28566.062,E2 -28566.062} C_VEL
LIN {X 0,Y 76.011,Z 428.536,A -85,B 0,C 180,E1 -28572.034,E2 -28572.034} C_VEL
LIN {X 0,Y 80.384,Z 421.579,A -85,B 0,C 180,E1 -28576.144,E2 -28576.144} C_VEL
LIN {X 0,Y 85.503,Z 412.17,A -85,B 0,C 180,E1 -28580.387,E2 -28580.387} C_VEL
LIN {X 0,Y 90.411,Z 401.916,A -85,B 0,C 180,E1 -28583.734,E2 -28583.734} C_VEL
LIN {X 0,Y 94.361,Z 392.546,A -85,B 0,C 180,E1 -28585.933,E2 -28585.933} C_VEL
LIN {X 0,Y 98.731,Z 379.479,A -85,B 0,C 180,E1 -28588.163,E2 -28588.163} C_VEL
LIN {X 0,Y 101.839,Z 366.938,A -85,B 0,C 180,E1 -28589.588,E2 -28589.588} C_VEL
LIN {X 0,Y 103.999,Z 353.251,A -85,B 0,C 180,E1 -28590.538,E2 -28590.538} C_VEL
LIN {X 0,Y 106.649,Z 323.907,A -85,B 0,C 180,E1 -28591.996,E2 -28591.996} C_VEL
LIN {X 0,Y 106.565,Z 320.114,A -85,B 0,C 180,E1 -28592.505,E2 -28592.505} C_VEL
LIN {X 0,Y 104.236,Z 311.435,A -85,B 0,C 180,E1 -28595.512,E2 -28595.512} C_VEL
LIN {X 0,Y 100.917,Z 304.58,A -85,B 0,C 180,E1 -28599.74,E2 -28599.74} C_VEL
LIN {X 0,Y 97.55,Z 298.435,A -85,B 0,C 180,E1 -28604.893,E2 -28604.893} C_VEL
LIN {X 0,Y 95.573,Z 295.051,A -85,B 0,C 180,E1 -28608.668,E2 -28608.668} C_VEL
LIN {X 0,Y 93.557,Z 291.606,A -85,B 0,C 180,E1 -28613.715,E2 -28613.715} C_VEL
LIN {X 0,Y 93.148,Z 290.756,A -85,B 0,C 180,E1 -28615.062,E2 -28615.062} C_VEL
LIN {X 0,Y 91.49,Z 288.23,A -85,B 0,C 180,E1 -28623.242,E2 -28623.242} C_VEL
LIN {X 0,Y 91.244,Z 288.375,A -85,B 0,C 180,E1 -28629.708,E2 -28629.708} C_VEL
LIN {X 0,Y 91.448,Z 289.289,A -85,B 0,C 180,E1 -28633.137,E2 -28633.137} C_VEL
LIN {X 0,Y 91.911,Z 290.972,A -85,B 0,C 180,E1 -28636.667,E2 -28636.667} C_VEL
LIN {X 0,Y 92.508,Z 293.71,A -85,B 0,C 180,E1 -28639.929,E2 -28639.929} C_VEL
LIN {X 0,Y 95.88,Z 305.359,A -85,B 0,C 180,E1 -28649.793,E2 -28649.793} C_VEL
LIN {X 0,Y 98.988,Z 311.559,A -85,B 0,C 180,E1 -28654.951,E2 -28654.951} C_VEL
LIN {X 0,Y 101.91,Z 318.286,A -85,B 0,C 180,E1 -28659.001,E2 -28659.001} C_VEL
LIN {X 0,Y 102.875,Z 320.839,A -85,B 0,C 180,E1 -28660.241,E2 -28660.241} C_VEL
LIN {X 0,Y 99.572,Z 352.739,A -85,B 0,C 180,E1 -28661.765,E2 -28661.765} C_VEL
LIN {X 0,Y 96.926,Z 366.415,A -85,B 0,C 180,E1 -28662.95,E2 -28662.95} C_VEL
LIN {X 0,Y 93.379,Z 379.156,A -85,B 0,C 180,E1 -28664.757,E2 -28664.757} C_VEL
LIN {X 0,Y 88.996,Z 390.872,A -85,B 0,C 180,E1 -28667.085,E2 -28667.085} C_VEL
LIN {X 0,Y 84.405,Z 400.892,A -85,B 0,C 180,E1 -28669.827,E2 -28669.827} C_VEL
LIN {X 0,Y 79.751,Z 409.925,A -85,B 0,C 180,E1 -28673.301,E2 -28673.301} C_VEL
LIN {X 0,Y 73.995,Z 419.488,A -85,B 0,C 180,E1 -28678.202,E2 -28678.202} C_VEL
LIN {X 0,Y 68.545,Z 427.724,A -85,B 0,C 180,E1 -28684.18,E2 -28684.18} C_VEL
LIN {X 0,Y 63.215,Z 435.418,A -85,B 0,C 180,E1 -28692.211,E2 -28692.211} C_VEL
LIN {X 0,Y 58.64,Z 442.532,A -85,B 0,C 180,E1 -28703.129,E2 -28703.129} C_VEL
LIN {X 0,Y 56.299,Z 447.028,A -85,B 0,C 180,E1 -28712.992,E2 -28712.992} C_VEL
LIN {X 0,Y 55.252,Z 450.914,A -85,B 0,C 180,E1 -28724.75,E2 -28724.75} C_VEL
LIN {X 0,Y 55.712,Z 452.737,A -85,B 0,C 180,E1 -28732.249,E2 -28732.249} C_VEL
LIN {X 0,Y 57.354,Z 454.367,A -85,B 0,C 180,E1 -28740.939,E2 -28740.939} C_VEL
LIN {X 0,Y 61.829,Z 455.67,A -85,B 0,C 180,E1 -28753.011,E2 -28753.011} C_VEL
LIN {X 0,Y 66.739,Z 455.739,A -85,B 0,C 180,E1 -28760.817,E2 -28760.817} C_VEL
LIN {X 0,Y 73.966,Z 454.768,A -85,B 0,C 180,E1 -28768.786,E2 -28768.786} C_VEL
LIN {X 0,Y 80.903,Z 453.043,A -85,B 0,C 180,E1 -28774.258,E2 -28774.258} C_VEL
LIN {X 0,Y 89.914,Z 449.893,A -85,B 0,C 180,E1 -28779.721,E2 -28779.721} C_VEL
LIN {X 0,Y 99.251,Z 445.57,A -85,B 0,C 180,E1 -28783.982,E2 -28783.982} C_VEL
LIN {X 0,Y 109.679,Z 439.426,A -85,B 0,C 180,E1 -28787.743,E2 -28787.743} C_VEL
LIN {X 0,Y 119.37,Z 432.383,A -85,B 0,C 180,E1 -28790.534,E2 -28790.534} C_VEL
LIN {X 0,Y 127.585,Z 425.148,A -85,B 0,C 180,E1 -28792.537,E2 -28792.537} C_VEL
LIN {X 0,Y 136.724,Z 415.374,A -85,B 0,C 180,E1 -28794.421,E2 -28794.421} C_VEL
LIN {X 0,Y 144.451,Z 405.236,A -85,B 0,C 180,E1 -28795.855,E2 -28795.855} C_VEL
LIN {X 0,Y 151.468,Z 393.771,A -85,B 0,C 180,E1 -28797.052,E2 -28797.052} C_VEL
LIN {X 0,Y 157.438,Z 381.178,A -85,B 0,C 180,E1 -28798.013,E2 -28798.013} C_VEL
LIN {X 0,Y 160.695,Z 372.387,A -85,B 0,C 180,E1 -28798.485,E2 -28798.485} C_VEL
LIN {X 0,Y 161.147,Z 370.882,A -85,B 0,C 180,E1 -28798.639,E2 -28798.639} C_VEL
LIN {X 0,Y 161.051,Z 369.68,A -85,B 0,C 180,E1 -28800.001,E2 -28800.001} C_VEL
LIN {X 0,Y 160.916,Z 366.335,A -85,B 0,C 180,E1 -28805.389,E2 -28805.389} C_VEL
LIN {X 0,Y 160.922,Z 366.409,A -85,B 0,C 180,E1 -28808.477,E2 -28808.477} C_VEL
LIN {X 0,Y 161.131,Z 369.525,A -85,B 0,C 180,E1 -28813.559,E2 -28813.559} C_VEL
LIN {X 0,Y 161.207,Z 371.735,A -85,B 0,C 180,E1 -28815.468,E2 -28815.468} C_VEL
LIN {X 0,Y 160.703,Z 373.679,A -85,B 0,C 180,E1 -28815.822,E2 -28815.822} C_VEL
LIN {X 0,Y 156.051,Z 385.948,A -85,B 0,C 180,E1 -28816.372,E2 -28816.372} C_VEL
LIN {X 0,Y 150.681,Z 396.815,A -85,B 0,C 180,E1 -28817.032,E2 -28817.032} C_VEL
LIN {X 0,Y 144.025,Z 407.547,A -85,B 0,C 180,E1 -28817.91,E2 -28817.91} C_VEL
LIN {X 0,Y 135.758,Z 418.301,A -85,B 0,C 180,E1 -28819.13,E2 -28819.13} C_VEL
LIN {X 0,Y 127.623,Z 427.05,A -85,B 0,C 180,E1 -28820.581,E2 -28820.581} C_VEL
LIN {X 0,Y 118.085,Z 435.596,A -85,B 0,C 180,E1 -28822.703,E2 -28822.703} C_VEL
LIN {X 0,Y 108.725,Z 442.472,A -85,B 0,C 180,E1 -28825.178,E2 -28825.178} C_VEL
LIN {X 0,Y 99.654,Z 448.013,A -85,B 0,C 180,E1 -28828.165,E2 -28828.165} C_VEL
LIN {X 0,Y 90.951,Z 452.396,A -85,B 0,C 180,E1 -28831.783,E2 -28831.783} C_VEL
LIN {X 0,Y 80.217,Z 456.66,A -85,B 0,C 180,E1 -28837.946,E2 -28837.946} C_VEL
LIN {X 0,Y 75.266,Z 458.152,A -85,B 0,C 180,E1 -28841.661,E2 -28841.661} C_VEL
LIN {X 0,Y 66.52,Z 459.944,A -85,B 0,C 180,E1 -28850.651,E2 -28850.651} C_VEL
LIN {X 0,Y 59.981,Z 460.24,A -85,B 0,C 180,E1 -28862.041,E2 -28862.041} C_VEL
LIN {X 0,Y 56.469,Z 458.96,A -85,B 0,C 180,E1 -28875.575,E2 -28875.575} C_VEL
LIN {X 0,Y 55.889,Z 457.744,A -85,B 0,C 180,E1 -28882.764,E2 -28882.764} C_VEL
LIN {X 0,Y 55.905,Z 456.111,A -85,B 0,C 180,E1 -28889.988,E2 -28889.988} C_VEL
LIN {X 0,Y 56.02,Z 452.67,A -85,B 0,C 180,E1 -28900.833,E2 -28900.833} C_VEL
LIN {X 0,Y 57.656,Z 448.085,A -85,B 0,C 180,E1 -28911.435,E2 -28911.435} C_VEL
LIN {X 0,Y 61.847,Z 441.111,A -85,B 0,C 180,E1 -28922.651,E2 -28922.651} C_VEL
LIN {X 0,Y 66.919,Z 433.511,A -85,B 0,C 180,E1 -28931.007,E2 -28931.007} C_VEL
LIN {X 0,Y 70.99,Z 427.29,A -85,B 0,C 180,E1 -28935.959,E2 -28935.959} C_VEL
LIN {X 0,Y 75.574,Z 420.296,A -85,B 0,C 180,E1 -28940.084,E2 -28940.084} C_VEL
LIN {X 0,Y 81.142,Z 410.694,A -85,B 0,C 180,E1 -28944.27,E2 -28944.27} C_VEL
LIN {X 0,Y 86.358,Z 400.182,A -85,B 0,C 180,E1 -28947.578,E2 -28947.578} C_VEL
LIN {X 0,Y 89.849,Z 392.267,A -85,B 0,C 180,E1 -28949.34,E2 -28949.34} C_VEL
LIN {X 0,Y 94.436,Z 379.216,A -85,B 0,C 180,E1 -28951.508,E2 -28951.508} C_VEL
LIN {X 0,Y 97.684,Z 366.682,A -85,B 0,C 180,E1 -28952.893,E2 -28952.893} C_VEL
LIN {X 0,Y 99.91,Z 353.236,A -85,B 0,C 180,E1 -28953.802,E2 -28953.802} C_VEL
LIN {X 0,Y 102.65,Z 324.544,A -85,B 0,C 180,E1 -28955.205,E2 -28955.205} C_VEL
LIN {X 0,Y 102.475,Z 322.003,A -85,B 0,C 180,E1 -28955.7,E2 -28955.7} C_VEL
LIN {X 0,Y 100.78,Z 315.557,A -85,B 0,C 180,E1 -28958.237,E2 -28958.237} C_VEL
LIN {X 0,Y 98.015,Z 309.53,A -85,B 0,C 180,E1 -28962.291,E2 -28962.291} C_VEL
LIN {X 0,Y 95.314,Z 304.226,A -85,B 0,C 180,E1 -28967.066,E2 -28967.066} C_VEL
LIN {X 0,Y 93.774,Z 301.358,A -85,B 0,C 180,E1 -28970.461,E2 -28970.461} C_VEL
LIN {X 0,Y 91.875,Z 297.564,A -85,B 0,C 180,E1 -28976.231,E2 -28976.231} C_VEL
LIN {X 0,Y 90.634,Z 295.388,A -85,B 0,C 180,E1 -28982.91,E2 -28982.91} C_VEL
LIN {X 0,Y 90.358,Z 295.491,A -85,B 0,C 180,E1 -28989.804,E2 -28989.804} C_VEL
LIN {X 0,Y 91.986,Z 298.266,A -85,B 0,C 180,E1 -29000.108,E2 -29000.108} C_VEL
LIN {X 0,Y 94.233,Z 302.416,A -85,B 0,C 180,E1 -29006.421,E2 -29006.421} C_VEL
LIN {X 0,Y 95.88,Z 305.359,A -85,B 0,C 180,E1 -29009.793,E2 -29009.793} C_VEL
LIN {X 0,Y 96.697,Z 307.964,A -85,B 0,C 180,E1 -29011.47,E2 -29011.47} C_VEL
LIN {X 0,Y 97.215,Z 311.259,A -85,B 0,C 180,E1 -29012.755,E2 -29012.755} C_VEL
LIN {X 0,Y 98.292,Z 320.896,A -85,B 0,C 180,E1 -29015.649,E2 -29015.649} C_VEL
LIN {X 0,Y 98.825,Z 323.047,A -85,B 0,C 180,E1 -29016.564,E2 -29016.564} C_VEL
LIN {X 0,Y 99.057,Z 323.683,A -85,B 0,C 180,E1 -29016.906,E2 -29016.906} C_VEL
LIN {X 0,Y 95.786,Z 353.359,A -85,B 0,C 180,E1 -29018.254,E2 -29018.254} C_VEL
LIN {X 0,Y 93.126,Z 366.476,A -85,B 0,C 180,E1 -29019.335,E2 -29019.335} C_VEL
LIN {X 0,Y 89.585,Z 378.776,A -85,B 0,C 180,E1 -29020.985,E2 -29020.985} C_VEL
LIN {X 0,Y 85.368,Z 389.821,A -85,B 0,C 180,E1 -29023.077,E2 -29023.077} C_VEL
LIN {X 0,Y 80.432,Z 400.115,A -85,B 0,C 180,E1 -29025.668,E2 -29025.668} C_VEL
LIN {X 0,Y 74.327,Z 411.203,A -85,B 0,C 180,E1 -29029.885,E2 -29029.885} C_VEL
LIN {X 0,Y 67.785,Z 421.14,A -85,B 0,C 180,E1 -29035.249,E2 -29035.249} C_VEL
LIN {X 0,Y 61.127,Z 430.216,A -85,B 0,C 180,E1 -29042.635,E2 -29042.635} C_VEL
LIN {X 0,Y 55.607,Z 437.527,A -85,B 0,C 180,E1 -29051.596,E2 -29051.596} C_VEL
LIN {X 0,Y 51.482,Z 443.368,A -85,B 0,C 180,E1 -29062.168,E2 -29062.168} C_VEL
LIN {X 0,Y 49.23,Z 447.342,A -85,B 0,C 180,E1 -29072.205,E2 -29072.205} C_VEL
LIN {X 0,Y 48.2,Z 451.526,A -85,B 0,C 180,E1 -29086.968,E2 -29086.968} C_VEL
LIN {X 0,Y 48.996,Z 453.287,A -85,B 0,C 180,E1 -29095.501,E2 -29095.501} C_VEL
LIN {X 0,Y 50.727,Z 454.65,A -85,B 0,C 180,E1 -29103.775,E2 -29103.775} C_VEL
LIN {X 0,Y 53.257,Z 455.567,A -85,B 0,C 180,E1 -29111.299,E2 -29111.299} C_VEL
LIN {X 0,Y 56.628,Z 456.035,A -85,B 0,C 180,E1 -29118.141,E2 -29118.141} C_VEL
LIN {X 0,Y 61.495,Z 456.077,A -85,B 0,C 180,E1 -29125.153,E2 -29125.153} C_VEL
LIN {X 0,Y 70.389,Z 454.954,A -85,B 0,C 180,E1 -29133.987,E2 -29133.987} C_VEL
LIN {X 0,Y 76.91,Z 453.444,A -85,B 0,C 180,E1 -29138.562,E2 -29138.562} C_VEL
LIN {X 0,Y 87.611,Z 449.888,A -85,B 0,C 180,E1 -29144.295,E2 -29144.295} C_VEL
LIN {X 0,Y 96.99,Z 445.695,A -85,B 0,C 180,E1 -29148.022,E2 -29148.022} C_VEL
LIN {X 0,Y 108.342,Z 439.193,A -85,B 0,C 180,E1 -29151.598,E2 -29151.598} C_VEL
LIN {X 0,Y 118.348,Z 432.001,A -85,B 0,C 180,E1 -29154.096,E2 -29154.096} C_VEL
LIN {X 0,Y 128.394,Z 423.057,A -85,B 0,C 180,E1 -29156.135,E2 -29156.135} C_VEL
LIN {X 0,Y 137.159,Z 413.496,A -85,B 0,C 180,E1 -29157.665,E2 -29157.665} C_VEL
LIN {X 0,Y 144.978,Z 402.889,A -85,B 0,C 180,E1 -29158.908,E2 -29158.908} C_VEL
LIN {X 0,Y 151.984,Z 390.982,A -85,B 0,C 180,E1 -29159.947,E2 -29159.947} C_VEL
LIN {X 0,Y 157.36,Z 379.187,A -85,B 0,C 180,E1 -29160.684,E2 -29160.684} C_VEL
LIN {X 0,Y 158.571,Z 375.899,A -85,B 0,C 180,E1 -29160.952,E2 -29160.952} C_VEL
LIN {X 0,Y 158.693,Z 373.475,A -85,B 0,C 180,E1 -29165.082,E2 -29165.082} C_VEL
LIN {X 0,Y 158.813,Z 372.994,A -85,B 0,C 180,E1 -29167.63,E2 -29167.63} C_VEL
LIN {X 0,Y 158.766,Z 376.22,A -85,B 0,C 180,E1 -29173.132,E2 -29173.132} C_VEL
LIN {X 0,Y 158.212,Z 377.949,A -85,B 0,C 180,E1 -29173.478,E2 -29173.478} C_VEL
LIN {X 0,Y 152.795,Z 390.496,A -85,B 0,C 180,E1 -29174.016,E2 -29174.016} C_VEL
LIN {X 0,Y 146.234,Z 402.191,A -85,B 0,C 180,E1 -29174.715,E2 -29174.715} C_VEL
LIN {X 0,Y 138.657,Z 412.912,A -85,B 0,C 180,E1 -29175.626,E2 -29175.626} C_VEL
LIN {X 0,Y 131.945,Z 420.81,A -85,B 0,C 180,E1 -29176.511,E2 -29176.511} C_VEL
LIN {X 0,Y 123.693,Z 429.042,A -85,B 0,C 180,E1 -29177.877,E2 -29177.877} C_VEL
LIN {X 0,Y 117.141,Z 434.656,A -85,B 0,C 180,E1 -29179.099,E2 -29179.099} C_VEL
LIN {X 0,Y 107.493,Z 441.653,A -85,B 0,C 180,E1 -29181.298,E2 -29181.298} C_VEL
LIN {X 0,Y 96.501,Z 448.101,A -85,B 0,C 180,E1 -29184.44,E2 -29184.44} C_VEL
LIN {X 0,Y 87.419,Z 452.388,A -85,B 0,C 180,E1 -29187.823,E2 -29187.823} C_VEL
LIN {X 0,Y 76.322,Z 456.464,A -85,B 0,C 180,E1 -29193.541,E2 -29193.541} C_VEL
LIN {X 0,Y 65.717,Z 459.008,A -85,B 0,C 180,E1 -29201.521,E2 -29201.521} C_VEL
LIN {X 0,Y 57.123,Z 459.969,A -85,B 0,C 180,E1 -29212.024,E2 -29212.024} C_VEL
LIN {X 0,Y 51.269,Z 459.364,A -85,B 0,C 180,E1 -29225.705,E2 -29225.705} C_VEL
LIN {X 0,Y 48.866,Z 457.241,A -85,B 0,C 180,E1 -29241.717,E2 -29241.717} C_VEL
LIN {X 0,Y 48.82,Z 455.539,A -85,B 0,C 180,E1 -29249.986,E2 -29249.986} C_VEL
LIN {X 0,Y 49.03,Z 452.013,A -85,B 0,C 180,E1 -29262.401,E2 -29262.401} C_VEL
LIN {X 0,Y 51.062,Z 447.324,A -85,B 0,C 180,E1 -29274.37,E2 -29274.37} C_VEL
LIN {X 0,Y 55.951,Z 440.233,A -85,B 0,C 180,E1 -29286.61,E2 -29286.61} C_VEL
LIN {X 0,Y 61.681,Z 432.508,A -85,B 0,C 180,E1 -29295.387,E2 -29295.387} C_VEL
LIN {X 0,Y 66.103,Z 426.365,A -85,B 0,C 180,E1 -29300.251,E2 -29300.251} C_VEL
LIN {X 0,Y 72.467,Z 417.024,A -85,B 0,C 180,E1 -29305.497,E2 -29305.497} C_VEL
LIN {X 0,Y 78.488,Z 406.716,A -85,B 0,C 180,E1 -29309.498,E2 -29309.498} C_VEL
LIN {X 0,Y 84.269,Z 395.335,A -85,B 0,C 180,E1 -29312.362,E2 -29312.362} C_VEL
LIN {X 0,Y 88.995,Z 383.436,A -85,B 0,C 180,E1 -29314.556,E2 -29314.556} C_VEL
LIN {X 0,Y 92.893,Z 370.567,A -85,B 0,C 180,E1 -29316.084,E2 -29316.084} C_VEL
LIN {X 0,Y 95.701,Z 356.939,A -85,B 0,C 180,E1 -29317.097,E2 -29317.097} C_VEL
LIN {X 0,Y 98.975,Z 326.058,A -85,B 0,C 180,E1 -29318.555,E2 -29318.555} C_VEL
LIN {X 0,Y 98.471,Z 322.945,A -85,B 0,C 180,E1 -29319.58,E2 -29319.58} C_VEL
LIN {X 0,Y 97.627,Z 319.948,A -85,B 0,C 180,E1 -29321.016,E2 -29321.016} C_VEL
LIN {X 0,Y 95.264,Z 314.38,A -85,B 0,C 180,E1 -29325.069,E2 -29325.069} C_VEL
LIN {X 0,Y 93.357,Z 310.281,A -85,B 0,C 180,E1 -29329.031,E2 -29329.031} C_VEL
LIN {X 0,Y 92.038,Z 307.576,A -85,B 0,C 180,E1 -29332.422,E2 -29332.422} C_VEL
LIN {X 0,Y 90.643,Z 304.372,A -85,B 0,C 180,E1 -29337.428,E2 -29337.428} C_VEL
LIN {X 0,Y 89.598,Z 302.268,A -85,B 0,C 180,E1 -29344.497,E2 -29344.497} C_VEL
LIN {X 0,Y 89.461,Z 302.697,A -85,B 0,C 180,E1 -29349.903,E2 -29349.903} C_VEL
LIN {X 0,Y 90.727,Z 305.019,A -85,B 0,C 180,E1 -29358.871,E2 -29358.871} C_VEL
LIN {X 0,Y 92.556,Z 308.83,A -85,B 0,C 180,E1 -29364.796,E2 -29364.796} C_VEL
LIN {X 0,Y 94.538,Z 312.914,A -85,B 0,C 180,E1 -29369.293,E2 -29369.293} C_VEL
LIN {X 0,Y 97.154,Z 318.778,A -85,B 0,C 180,E1 -29373.978,E2 -29373.978} C_VEL
LIN {X 0,Y 98.825,Z 323.047,A -85,B 0,C 180,E1 -29376.564,E2 -29376.564} C_VEL
LIN {X 0,Y 99.211,Z 325.401,A -85,B 0,C 180,E1 -29377.309,E2 -29377.309} C_VEL
LIN {X 0,Y 99.082,Z 329.029,A -85,B 0,C 180,E1 -29377.667,E2 -29377.667} C_VEL
LIN {X 0,Y 98.199,Z 333.789,A -85,B 0,C 180,E1 -29377.395,E2 -29377.395} C_VEL
LIN {X 0,Y 97.155,Z 337.469,A -85,B 0,C 180,E1 -29376.813,E2 -29376.813} C_VEL
LIN {X 0,Y 93.874,Z 347.499,A -85,B 0,C 180,E1 -29374.811,E2 -29374.811} C_VEL
LIN {X 0,Y 92.573,Z 352.736,A -85,B 0,C 180,E1 -29374.432,E2 -29374.432} C_VEL
LIN {X 0,Y 92.375,Z 353.802,A -85,B 0,C 180,E1 -29374.475,E2 -29374.475} C_VEL
LIN {X 0,Y 89.499,Z 367.276,A -85,B 0,C 180,E1 -29375.516,E2 -29375.516} C_VEL
LIN {X 0,Y 85.841,Z 379.283,A -85,B 0,C 180,E1 -29377.056,E2 -29377.056} C_VEL
LIN {X 0,Y 81.413,Z 390.29,A -85,B 0,C 180,E1 -29379.04,E2 -29379.04} C_VEL
LIN {X 0,Y 76.217,Z 400.559,A -85,B 0,C 180,E1 -29381.498,E2 -29381.498} C_VEL
LIN {X 0,Y 70.036,Z 411.125,A -85,B 0,C 180,E1 -29385.397,E2 -29385.397} C_VEL
LIN {X 0,Y 63.336,Z 420.709,A -85,B 0,C 180,E1 -29390.373,E2 -29390.373} C_VEL
LIN {X 0,Y 56.014,Z 429.918,A -85,B 0,C 180,E1 -29397.794,E2 -29397.794} C_VEL
LIN {X 0,Y 49.762,Z 437.341,A -85,B 0,C 180,E1 -29407.163,E2 -29407.163} C_VEL
LIN {X 0,Y 45.66,Z 442.374,A -85,B 0,C 180,E1 -29416.668,E2 -29416.668} C_VEL
LIN {X 0,Y 42.173,Z 447.615,A -85,B 0,C 180,E1 -29431.089,E2 -29431.089} C_VEL
LIN {X 0,Y 41.067,Z 451.086,A -85,B 0,C 180,E1 -29444.891,E2 -29444.891} C_VEL
LIN {X 0,Y 42.451,Z 453.832,A -85,B 0,C 180,E1 -29459.796,E2 -29459.796} C_VEL
LIN {X 0,Y 44.723,Z 455.136,A -85,B 0,C 180,E1 -29468.961,E2 -29468.961} C_VEL
LIN {X 0,Y 47.939,Z 455.977,A -85,B 0,C 180,E1 -29477.155,E2 -29477.155} C_VEL
LIN {X 0,Y 51.96,Z 456.4,A -85,B 0,C 180,E1 -29484.263,E2 -29484.263} C_VEL
LIN {X 0,Y 56.667,Z 456.416,A -85,B 0,C 180,E1 -29490.261,E2 -29490.261} C_VEL
LIN {X 0,Y 61.861,Z 456.007,A -85,B 0,C 180,E1 -29495.366,E2 -29495.366} C_VEL
LIN {X 0,Y 67.46,Z 455.136,A -85,B 0,C 180,E1 -29499.671,E2 -29499.671} C_VEL
LIN {X 0,Y 73.379,Z 453.848,A -85,B 0,C 180,E1 -29503.304,E2 -29503.304} C_VEL
LIN {X 0,Y 82.694,Z 451.052,A -85,B 0,C 180,E1 -29507.802,E2 -29507.802} C_VEL
LIN {X 0,Y 92.415,Z 447.151,A -85,B 0,C 180,E1 -29511.365,E2 -29511.365} C_VEL
LIN {X 0,Y 102.425,Z 442.029,A -85,B 0,C 180,E1 -29514.244,E2 -29514.244} C_VEL
LIN {X 0,Y 112.644,Z 435.477,A -85,B 0,C 180,E1 -29516.639,E2 -29516.639} C_VEL
LIN {X 0,Y 123.027,Z 427.206,A -85,B 0,C 180,E1 -29518.603,E2 -29518.603} C_VEL
LIN {X 0,Y 131.797,Z 418.668,A -85,B 0,C 180,E1 -29520.001,E2 -29520.001} C_VEL
LIN {X 0,Y 139.708,Z 409.314,A -85,B 0,C 180,E1 -29521.131,E2 -29521.131} C_VEL
LIN {X 0,Y 146.802,Z 398.981,A -85,B 0,C 180,E1 -29522.053,E2 -29522.053} C_VEL
LIN {X 0,Y 153.12,Z 387.451,A -85,B 0,C 180,E1 -29522.853,E2 -29522.853} C_VEL
LIN {X 0,Y 155.818,Z 381.502,A -85,B 0,C 180,E1 -29523.168,E2 -29523.168} C_VEL
LIN {X 0,Y 156.157,Z 380.186,A -85,B 0,C 180,E1 -29525.165,E2 -29525.165} C_VEL
LIN {X 0,Y 156.288,Z 379.827,A -85,B 0,C 180,E1 -29527.754,E2 -29527.754} C_VEL
LIN {X 0,Y 156.083,Z 381.219,A -85,B 0,C 180,E1 -29530.377,E2 -29530.377} C_VEL
LIN {X 0,Y 155.67,Z 382.493,A -85,B 0,C 180,E1 -29531.053,E2 -29531.053} C_VEL
LIN {X 0,Y 149.747,Z 394.679,A -85,B 0,C 180,E1 -29531.563,E2 -29531.563} C_VEL
LIN {X 0,Y 142.898,Z 405.758,A -85,B 0,C 180,E1 -29532.181,E2 -29532.181} C_VEL
LIN {X 0,Y 135.218,Z 415.752,A -85,B 0,C 180,E1 -29532.958,E2 -29532.958} C_VEL
LIN {X 0,Y 126.757,Z 424.812,A -85,B 0,C 180,E1 -29534.003,E2 -29534.003} C_VEL
LIN {X 0,Y 116.657,Z 433.679,A -85,B 0,C 180,E1 -29535.434,E2 -29535.434} C_VEL
LIN {X 0,Y 106.771,Z 440.823,A -85,B 0,C 180,E1 -29537.358,E2 -29537.358} C_VEL
LIN {X 0,Y 97,Z 446.564,A -85,B 0,C 180,E1 -29539.621,E2 -29539.621} C_VEL
LIN {X 0,Y 87.453,Z 451.122,A -85,B 0,C 180,E1 -29542.448,E2 -29542.448} C_VEL
LIN {X 0,Y 78.251,Z 454.625,A -85,B 0,C 180,E1 -29546.076,E2 -29546.076} C_VEL
LIN {X 0,Y 66.648,Z 457.785,A -85,B 0,C 180,E1 -29552.467,E2 -29552.467} C_VEL
LIN {X 0,Y 56.238,Z 459.411,A -85,B 0,C 180,E1 -29561.413,E2 -29561.413} C_VEL
LIN {X 0,Y 47.844,Z 459.464,A -85,B 0,C 180,E1 -29574,E2 -29574} C_VEL
LIN {X 0,Y 42.84,Z 458.025,A -85,B 0,C 180,E1 -29590.831,E2 -29590.831} C_VEL
LIN {X 0,Y 41.844,Z 456.723,A -85,B 0,C 180,E1 -29600.315,E2 -29600.315} C_VEL
LIN {X 0,Y 41.736,Z 454.949,A -85,B 0,C 180,E1 -29609.983,E2 -29609.983} C_VEL
LIN {X 0,Y 42.103,Z 451.333,A -85,B 0,C 180,E1 -29624.482,E2 -29624.482} C_VEL
LIN {X 0,Y 44.65,Z 446.545,A -85,B 0,C 180,E1 -29638.157,E2 -29638.157} C_VEL
LIN {X 0,Y 50.388,Z 439.347,A -85,B 0,C 180,E1 -29651.469,E2 -29651.469} C_VEL
LIN {X 0,Y 56.846,Z 431.437,A -85,B 0,C 180,E1 -29660.572,E2 -29660.572} C_VEL
LIN {X 0,Y 61.996,Z 424.995,A -85,B 0,C 180,E1 -29665.47,E2 -29665.47} C_VEL
LIN {X 0,Y 68.64,Z 415.643,A -85,B 0,C 180,E1 -29670.465,E2 -29670.465} C_VEL
LIN {X 0,Y 75.128,Z 405.095,A -85,B 0,C 180,E1 -29674.177,E2 -29674.177} C_VEL
LIN {X 0,Y 81.189,Z 393.407,A -85,B 0,C 180,E1 -29676.853,E2 -29676.853} C_VEL
LIN {X 0,Y 85.762,Z 382.021,A -85,B 0,C 180,E1 -29678.737,E2 -29678.737} C_VEL
LIN {X 0,Y 89.701,Z 369.28,A -85,B 0,C 180,E1 -29680.047,E2 -29680.047} C_VEL
LIN {X 0,Y 92.433,Z 356.027,A -85,B 0,C 180,E1 -29680.968,E2 -29680.968} C_VEL
LIN {X 0,Y 95.557,Z 327.705,A -85,B 0,C 180,E1 -29682.218,E2 -29682.218} C_VEL
LIN {X 0,Y 94.879,Z 324.87,A -85,B 0,C 180,E1 -29683.612,E2 -29683.612} C_VEL
LIN {X 0,Y 92.963,Z 319.773,A -85,B 0,C 180,E1 -29687.52,E2 -29687.52} C_VEL
LIN {X 0,Y 91.484,Z 316.255,A -85,B 0,C 180,E1 -29691.16,E2 -29691.16} C_VEL
LIN {X 0,Y 90.587,Z 314.166,A -85,B 0,C 180,E1 -29693.875,E2 -29693.875} C_VEL
LIN {X 0,Y 89.405,Z 311.069,A -85,B 0,C 180,E1 -29698.903,E2 -29698.903} C_VEL
LIN {X 0,Y 88.708,Z 309.341,A -85,B 0,C 180,E1 -29704.543,E2 -29704.543} C_VEL
LIN {X 0,Y 88.566,Z 309.732,A -85,B 0,C 180,E1 -29709.567,E2 -29709.567} C_VEL
LIN {X 0,Y 89.559,Z 311.89,A -85,B 0,C 180,E1 -29717.837,E2 -29717.837} C_VEL
LIN {X 0,Y 91.017,Z 315.365,A -85,B 0,C 180,E1 -29723.294,E2 -29723.294} C_VEL
LIN {X 0,Y 92.889,Z 319.648,A -85,B 0,C 180,E1 -29728.074,E2 -29728.074} C_VEL
LIN {X 0,Y 95.173,Z 325.686,A -85,B 0,C 180,E1 -29732.681,E2 -29732.681} C_VEL
LIN {X 0,Y 95.518,Z 326.591,A -85,B 0,C 180,E1 -29733.29,E2 -29733.29} C_VEL
LIN {X 0,Y 92.375,Z 353.802,A -85,B 0,C 180,E1 -29734.475,E2 -29734.475} C_VEL
LIN {X 0,Y 91.383,Z 357.67,A -85,B 0,C 180,E1 -29734.308,E2 -29734.308} C_VEL
LIN {X 0,Y 86.114,Z 369.581,A -85,B 0,C 180,E1 -29731.918,E2 -29731.918} C_VEL
LIN {X 0,Y 84.77,Z 373.322,A -85,B 0,C 180,E1 -29731.988,E2 -29731.988} C_VEL
LIN {X 0,Y 80.256,Z 385.572,A -85,B 0,C 180,E1 -29733.728,E2 -29733.728} C_VEL
LIN {X 0,Y 74.708,Z 396.897,A -85,B 0,C 180,E1 -29735.792,E2 -29735.792} C_VEL
LIN {X 0,Y 68.795,Z 407.134,A -85,B 0,C 180,E1 -29738.857,E2 -29738.857} C_VEL
LIN {X 0,Y 62.422,Z 416.37,A -85,B 0,C 180,E1 -29742.738,E2 -29742.738} C_VEL
LIN {X 0,Y 55.308,Z 425.2,A -85,B 0,C 180,E1 -29748.177,E2 -29748.177} C_VEL
LIN {X 0,Y 47.674,Z 433.586,A -85,B 0,C 180,E1 -29756.46,E2 -29756.46} C_VEL
LIN {X 0,Y 41.267,Z 440.347,A -85,B 0,C 180,E1 -29767.489,E2 -29767.489} C_VEL
LIN {X 0,Y 36.082,Z 446.478,A -85,B 0,C 180,E1 -29784.189,E2 -29784.189} C_VEL
LIN {X 0,Y 33.998,Z 450.606,A -85,B 0,C 180,E1 -29801.95,E2 -29801.95} C_VEL
LIN {X 0,Y 34.405,Z 452.706,A -85,B 0,C 180,E1 -29814.133,E2 -29814.133} C_VEL
LIN {X 0,Y 38.05,Z 455.209,A -85,B 0,C 180,E1 -29832.374,E2 -29832.374} C_VEL
LIN {X 0,Y 43.23,Z 456.387,A -85,B 0,C 180,E1 -29844.397,E2 -29844.397} C_VEL
LIN {X 0,Y 52.361,Z 456.755,A -85,B 0,C 180,E1 -29856.258,E2 -29856.258} C_VEL
LIN {X 0,Y 59.144,Z 456.235,A -85,B 0,C 180,E1 -29861.942,E2 -29861.942} C_VEL
LIN {X 0,Y 70.422,Z 454.247,A -85,B 0,C 180,E1 -29868.489,E2 -29868.489} C_VEL
LIN {X 0,Y 81.447,Z 451.092,A -85,B 0,C 180,E1 -29872.925,E2 -29872.925} C_VEL
LIN {X 0,Y 91.595,Z 447.086,A -85,B 0,C 180,E1 -29875.963,E2 -29875.963} C_VEL
LIN {X 0,Y 103.689,Z 440.794,A -85,B 0,C 180,E1 -29878.79,E2 -29878.79} C_VEL
LIN {X 0,Y 114.216,Z 433.852,A -85,B 0,C 180,E1 -29880.718,E2 -29880.718} C_VEL
LIN {X 0,Y 123.07,Z 426.702,A -85,B 0,C 180,E1 -29882.059,E2 -29882.059} C_VEL
LIN {X 0,Y 131.823,Z 418.175,A -85,B 0,C 180,E1 -29883.179,E2 -29883.179} C_VEL
LIN {X 0,Y 140.049,Z 408.331,A -85,B 0,C 180,E1 -29884.158,E2 -29884.158} C_VEL
LIN {X 0,Y 147.252,Z 397.705,A -85,B 0,C 180,E1 -29884.926,E2 -29884.926} C_VEL
LIN {X 0,Y 153.255,Z 386.615,A -85,B 0,C 180,E1 -29885.593,E2 -29885.593} C_VEL
LIN {X 0,Y 153.366,Z 386.513,A -85,B 0,C 180,E1 -29887.903,E2 -29887.903} C_VEL
LIN {X 0,Y 152.772,Z 387.854,A -85,B 0,C 180,E1 -29888.598,E2 -29888.598} C_VEL
LIN {X 0,Y 145.898,Z 400.252,A -85,B 0,C 180,E1 -29889.072,E2 -29889.072} C_VEL
LIN {X 0,Y 138.12,Z 411.257,A -85,B 0,C 180,E1 -29889.646,E2 -29889.646} C_VEL
LIN {X 0,Y 128.65,Z 421.984,A -85,B 0,C 180,E1 -29890.479,E2 -29890.479} C_VEL
LIN {X 0,Y 120.106,Z 429.916,A -85,B 0,C 180,E1 -29891.44,E2 -29891.44} C_VEL
LIN {X 0,Y 113.294,Z 435.287,A -85,B 0,C 180,E1 -29892.3,E2 -29892.3} C_VEL
LIN {X 0,Y 101.519,Z 443.047,A -85,B 0,C 180,E1 -29894.251,E2 -29894.251} C_VEL
LIN {X 0,Y 91.539,Z 448.278,A -85,B 0,C 180,E1 -29896.313,E2 -29896.313} C_VEL
LIN {X 0,Y 81.753,Z 452.373,A -85,B 0,C 180,E1 -29898.971,E2 -29898.971} C_VEL
LIN {X 0,Y 75.391,Z 454.538,A -85,B 0,C 180,E1 -29901.207,E2 -29901.207} C_VEL
LIN {X 0,Y 63.108,Z 457.602,A -85,B 0,C 180,E1 -29906.997,E2 -29906.997} C_VEL
LIN {X 0,Y 51.795,Z 459.125,A -85,B 0,C 180,E1 -29915.482,E2 -29915.482} C_VEL
LIN {X 0,Y 42.282,Z 459.073,A -85,B 0,C 180,E1 -29928.311,E2 -29928.311} C_VEL
LIN {X 0,Y 36.189,Z 457.55,A -85,B 0,C 180,E1 -29947.126,E2 -29947.126} C_VEL
LIN {X 0,Y 34.875,Z 456.17,A -85,B 0,C 180,E1 -29958.355,E2 -29958.355} C_VEL
LIN {X 0,Y 34.626,Z 454.346,A -85,B 0,C 180,E1 -29969.98,E2 -29969.98} C_VEL
LIN {X 0,Y 35.242,Z 450.635,A -85,B 0,C 180,E1 -29987.383,E2 -29987.383} C_VEL
LIN {X 0,Y 38.506,Z 445.747,A -85,B 0,C 180,E1 -30003.174,E2 -30003.174} C_VEL
LIN {X 0,Y 44.172,Z 439.571,A -85,B 0,C 180,E1 -30015.695,E2 -30015.695} C_VEL
LIN {X 0,Y 51.293,Z 431.837,A -85,B 0,C 180,E1 -30025.264,E2 -30025.264} C_VEL
LIN {X 0,Y 56.692,Z 425.591,A -85,B 0,C 180,E1 -30030.167,E2 -30030.167} C_VEL
LIN {X 0,Y 63.935,Z 416.346,A -85,B 0,C 180,E1 -30035.04,E2 -30035.04} C_VEL
LIN {X 0,Y 69.975,Z 407.317,A -85,B 0,C 180,E1 -30038.245,E2 -30038.245} C_VEL
LIN {X 0,Y 76.259,Z 396.218,A -85,B 0,C 180,E1 -30040.802,E2 -30040.802} C_VEL
LIN {X 0,Y 81.446,Z 384.742,A -85,B 0,C 180,E1 -30042.621,E2 -30042.621} C_VEL
LIN {X 0,Y 85.897,Z 371.883,A -85,B 0,C 180,E1 -30043.975,E2 -30043.975} C_VEL
LIN {X 0,Y 88.875,Z 359.308,A -85,B 0,C 180,E1 -30044.843,E2 -30044.843} C_VEL
LIN {X 0,Y 91.292,Z 341.012,A -85,B 0,C 180,E1 -30045.625,E2 -30045.625} C_VEL
LIN {X 0,Y 92.439,Z 330.138,A -85,B 0,C 180,E1 -30046.12,E2 -30046.12} C_VEL
LIN {X 0,Y 90.876,Z 325.335,A -85,B 0,C 180,E1 -30049.978,E2 -30049.978} C_VEL
LIN {X 0,Y 89.404,Z 321.125,A -85,B 0,C 180,E1 -30054.642,E2 -30054.642} C_VEL
LIN {X 0,Y 88.298,Z 317.885,A -85,B 0,C 180,E1 -30059.999,E2 -30059.999} C_VEL
LIN {X 0,Y 87.813,Z 316.456,A -85,B 0,C 180,E1 -30064.589,E2 -30064.589} C_VEL
LIN {X 0,Y 87.674,Z 316.685,A -85,B 0,C 180,E1 -30068.816,E2 -30068.816} C_VEL
LIN {X 0,Y 88.406,Z 318.737,A -85,B 0,C 180,E1 -30076.699,E2 -30076.699} C_VEL
LIN {X 0,Y 89.549,Z 321.902,A -85,B 0,C 180,E1 -30081.755,E2 -30081.755} C_VEL
LIN {X 0,Y 90.976,Z 325.719,A -85,B 0,C 180,E1 -30086.062,E2 -30086.062} C_VEL
LIN {X 0,Y 92.36,Z 329.836,A -85,B 0,C 180,E1 -30089.44,E2 -30089.44} C_VEL
LIN {X 0,Y 89.381,Z 354.323,A -85,B 0,C 180,E1 -30090.43,E2 -30090.43} C_VEL
LIN {X 0,Y 86.387,Z 367.759,A -85,B 0,C 180,E1 -30091.37,E2 -30091.37} C_VEL
LIN {X 0,Y 84.77,Z 373.322,A -85,B 0,C 180,E1 -30091.988,E2 -30091.988} C_VEL
LIN {X 0,Y 83.504,Z 377.029,A -85,B 0,C 180,E1 -30092.287,E2 -30092.287} C_VEL
LIN {X 0,Y 81.011,Z 382.418,A -85,B 0,C 180,E1 -30092.146,E2 -30092.146} C_VEL
LIN {X 0,Y 73.774,Z 394.276,A -85,B 0,C 180,E1 -30091.032,E2 -30091.032} C_VEL
LIN {X 0,Y 70.555,Z 399.254,A -85,B 0,C 180,E1 -30091.291,E2 -30091.291} C_VEL
LIN {X 0,Y 69.537,Z 400.9,A -85,B 0,C 180,E1 -30091.627,E2 -30091.627} C_VEL
LIN {X 0,Y 62.261,Z 411.966,A -85,B 0,C 180,E1 -30095.105,E2 -30095.105} C_VEL
LIN {X 0,Y 54.612,Z 421.511,A -85,B 0,C 180,E1 -30099.481,E2 -30099.481} C_VEL
LIN {X 0,Y 45.944,Z 430.689,A -85,B 0,C 180,E1 -30106.525,E2 -30106.525} C_VEL
LIN {X 0,Y 38.12,Z 438.097,A -85,B 0,C 180,E1 -30116.446,E2 -30116.446} C_VEL
LIN {X 0,Y 31.828,Z 444.033,A -85,B 0,C 180,E1 -30130.682,E2 -30130.682} C_VEL
LIN {X 0,Y 27.743,Z 448.743,A -85,B 0,C 180,E1 -30150.025,E2 -30150.025} C_VEL
LIN {X 0,Y 27.155,Z 452.348,A -85,B 0,C 180,E1 -30172.869,E2 -30172.869} C_VEL
LIN {X 0,Y 32.217,Z 455.488,A -85,B 0,C 180,E1 -30199.128,E2 -30199.128} C_VEL
LIN {X 0,Y 39.365,Z 456.798,A -85,B 0,C 180,E1 -30213.24,E2 -30213.24} C_VEL
LIN {X 0,Y 48.674,Z 457.096,A -85,B 0,C 180,E1 -30223.218,E2 -30223.218} C_VEL
LIN {X 0,Y 57.275,Z 456.463,A -85,B 0,C 180,E1 -30229.042,E2 -30229.042} C_VEL
LIN {X 0,Y 68.077,Z 454.649,A -85,B 0,C 180,E1 -30234.076,E2 -30234.076} C_VEL
LIN {X 0,Y 80.869,Z 451.112,A -85,B 0,C 180,E1 -30238.155,E2 -30238.155} C_VEL
LIN {X 0,Y 91.373,Z 446.987,A -85,B 0,C 180,E1 -30240.604,E2 -30240.604} C_VEL
LIN {X 0,Y 103.796,Z 440.563,A -85,B 0,C 180,E1 -30242.878,E2 -30242.878} C_VEL
LIN {X 0,Y 114.545,Z 433.491,A -85,B 0,C 180,E1 -30244.403,E2 -30244.403} C_VEL
LIN {X 0,Y 123.554,Z 426.184,A -85,B 0,C 180,E1 -30245.47,E2 -30245.47} C_VEL
LIN {X 0,Y 133.151,Z 416.626,A -85,B 0,C 180,E1 -30246.427,E2 -30246.427} C_VEL
LIN {X 0,Y 134.409,Z 415.232,A -85,B 0,C 180,E1 -30246.551,E2 -30246.551} C_VEL
LIN {X 0,Y 134.506,Z 415.153,A -85,B 0,C 180,E1 -30246.901,E2 -30246.901} C_VEL
LIN {X 0,Y 125.827,Z 424.207,A -85,B 0,C 180,E1 -30247.509,E2 -30247.509} C_VEL
LIN {X 0,Y 115.449,Z 433.06,A -85,B 0,C 180,E1 -30248.413,E2 -30248.413} C_VEL
LIN {X 0,Y 105.14,Z 440.198,A -85,B 0,C 180,E1 -30249.605,E2 -30249.605} C_VEL
LIN {X 0,Y 93.195,Z 446.741,A -85,B 0,C 180,E1 -30251.364,E2 -30251.364} C_VEL
LIN {X 0,Y 83.073,Z 451.108,A -85,B 0,C 180,E1 -30253.354,E2 -30253.354} C_VEL
LIN {X 0,Y 73.113,Z 454.44,A -85,B 0,C 180,E1 -30255.986,E2 -30255.986} C_VEL
LIN {X 0,Y 60.209,Z 457.419,A -85,B 0,C 180,E1 -30260.944,E2 -30260.944} C_VEL
LIN {X 0,Y 53.991,Z 458.327,A -85,B 0,C 180,E1 -30264.31,E2 -30264.31} C_VEL
LIN {X 0,Y 42.397,Z 458.935,A -85,B 0,C 180,E1 -30274,E2 -30274} C_VEL
LIN {X 0,Y 32.981,Z 458.068,A -85,B 0,C 180,E1 -30290.239,E2 -30290.239} C_VEL
LIN {X 0,Y 29.766,Z 457.051,A -85,B 0,C 180,E1 -30301.798,E2 -30301.798} C_VEL
LIN {X 0,Y 27.958,Z 455.612,A -85,B 0,C 180,E1 -30315.417,E2 -30315.417} C_VEL
LIN {X 0,Y 27.536,Z 453.745,A -85,B 0,C 180,E1 -30329.975,E2 -30329.975} C_VEL
LIN {X 0,Y 28.522,Z 449.937,A -85,B 0,C 180,E1 -30351.663,E2 -30351.663} C_VEL
LIN {X 0,Y 32.756,Z 444.948,A -85,B 0,C 180,E1 -30370.033,E2 -30370.033} C_VEL
LIN {X 0,Y 39.505,Z 438.661,A -85,B 0,C 180,E1 -30383.147,E2 -30383.147} C_VEL
LIN {X 0,Y 47.558,Z 430.737,A -85,B 0,C 180,E1 -30392.415,E2 -30392.415} C_VEL
LIN {X 0,Y 54.906,Z 422.853,A -85,B 0,C 180,E1 -30397.589,E2 -30397.589} C_VEL
LIN {X 0,Y 62.054,Z 413.855,A -85,B 0,C 180,E1 -30401.483,E2 -30401.483} C_VEL
LIN {X 0,Y 69.289,Z 403.071,A -85,B 0,C 180,E1 -30404.434,E2 -30404.434} C_VEL
LIN {X 0,Y 75.046,Z 392.653,A -85,B 0,C 180,E1 -30406.253,E2 -30406.253} C_VEL
LIN {X 0,Y 80.278,Z 380.511,A -85,B 0,C 180,E1 -30407.748,E2 -30407.748} C_VEL
LIN {X 0,Y 84.329,Z 367.905,A -85,B 0,C 180,E1 -30408.736,E2 -30408.736} C_VEL
LIN {X 0,Y 86.96,Z 355.881,A -85,B 0,C 180,E1 -30409.361,E2 -30409.361} C_VEL
LIN {X 0,Y 89.71,Z 333.494,A -85,B 0,C 180,E1 -30410.168,E2 -30410.168} C_VEL
LIN {X 0,Y 88.304,Z 328.702,A -85,B 0,C 180,E1 -30415.005,E2 -30415.005} C_VEL
LIN {X 0,Y 87.258,Z 324.838,A -85,B 0,C 180,E1 -30420.834,E2 -30420.834} C_VEL
LIN {X 0,Y 86.91,Z 323.632,A -85,B 0,C 180,E1 -30424.637,E2 -30424.637} C_VEL
LIN {X 0,Y 86.781,Z 323.761,A -85,B 0,C 180,E1 -30428.496,E2 -30428.496} C_VEL
LIN {X 0,Y 87.314,Z 325.671,A -85,B 0,C 180,E1 -30435.712,E2 -30435.712} C_VEL
LIN {X 0,Y 88.131,Z 328.427,A -85,B 0,C 180,E1 -30440.113,E2 -30440.113} C_VEL
LIN {X 0,Y 89.181,Z 331.802,A -85,B 0,C 180,E1 -30443.974,E2 -30443.974} C_VEL
LIN {X 0,Y 89.609,Z 333.336,A -85,B 0,C 180,E1 -30445.329,E2 -30445.329} C_VEL
LIN {X 0,Y 86.801,Z 355.231,A -85,B 0,C 180,E1 -30446.163,E2 -30446.163} C_VEL
LIN {X 0,Y 83.871,Z 367.811,A -85,B 0,C 180,E1 -30446.9,E2 -30446.9} C_VEL
LIN {X 0,Y 79.732,Z 380.279,A -85,B 0,C 180,E1 -30448.211,E2 -30448.211} C_VEL
LIN {X 0,Y 74.886,Z 391.225,A -85,B 0,C 180,E1 -30449.789,E2 -30449.789} C_VEL
LIN {X 0,Y 69.537,Z 400.9,A -85,B 0,C 180,E1 -30451.627,E2 -30451.627} C_VEL
LIN {X 0,Y 66.237,Z 405.785,A -85,B 0,C 180,E1 -30452.416,E2 -30452.416} C_VEL
LIN {X 0,Y 59.782,Z 413.32,A -85,B 0,C 180,E1 -30452.436,E2 -30452.436} C_VEL
LIN {X 0,Y 52.809,Z 420.385,A -85,B 0,C 180,E1 -30452.667,E2 -30452.667} C_VEL
LIN {X 0,Y 48.728,Z 424.445,A -85,B 0,C 180,E1 -30454.157,E2 -30454.157} C_VEL
LIN {X 0,Y 41.041,Z 431.763,A -85,B 0,C 180,E1 -30459.626,E2 -30459.626} C_VEL
LIN {X 0,Y 32.39,Z 439.033,A -85,B 0,C 180,E1 -30469.42,E2 -30469.42} C_VEL
LIN {X 0,Y 25.115,Z 444.828,A -85,B 0,C 180,E1 -30485.214,E2 -30485.214} C_VEL
LIN {X 0,Y 20.428,Z 449.431,A -85,B 0,C 180,E1 -30510.034,E2 -30510.034} C_VEL
LIN {X 0,Y 20.578,Z 452.941,A -85,B 0,C 180,E1 -30540.852,E2 -30540.852} C_VEL
LIN {X 0,Y 27.037,Z 455.77,A -85,B 0,C 180,E1 -30568.682,E2 -30568.682} C_VEL
LIN {X 0,Y 36.621,Z 457.21,A -85,B 0,C 180,E1 -30583.697,E2 -30583.697} C_VEL
LIN {X 0,Y 45.839,Z 457.436,A -85,B 0,C 180,E1 -30591.183,E2 -30591.183} C_VEL
LIN {X 0,Y 56.335,Z 456.692,A -85,B 0,C 180,E1 -30596.515,E2 -30596.515} C_VEL
LIN {X 0,Y 66.429,Z 455.049,A -85,B 0,C 180,E1 -30600.002,E2 -30600.002} C_VEL
LIN {X 0,Y 80.972,Z 451.101,A -85,B 0,C 180,E1 -30603.433,E2 -30603.433} C_VEL
LIN {X 0,Y 93.895,Z 445.892,A -85,B 0,C 180,E1 -30605.575,E2 -30605.575} C_VEL
LIN {X 0,Y 96.04,Z 444.866,A -85,B 0,C 180,E1 -30605.879,E2 -30605.879} C_VEL
LIN {X 0,Y 92.06,Z 446.83,A -85,B 0,C 180,E1 -30607.031,E2 -30607.031} C_VEL
LIN {X 0,Y 81.725,Z 451.101,A -85,B 0,C 180,E1 -30608.501,E2 -30608.501} C_VEL
LIN {X 0,Y 71.479,Z 454.342,A -85,B 0,C 180,E1 -30610.484,E2 -30610.484} C_VEL
LIN {X 0,Y 58.045,Z 457.234,A -85,B 0,C 180,E1 -30614.362,E2 -30614.362} C_VEL
LIN {X 0,Y 45.039,Z 458.509,A -85,B 0,C 180,E1 -30620.538,E2 -30620.538} C_VEL
LIN {X 0,Y 33.028,Z 458.292,A -85,B 0,C 180,E1 -30631.629,E2 -30631.629} C_VEL
LIN {X 0,Y 27.874,Z 457.623,A -85,B 0,C 180,E1 -30640.819,E2 -30640.819} C_VEL
LIN {X 0,Y 23.744,Z 456.536,A -85,B 0,C 180,E1 -30653.67,E2 -30653.67} C_VEL
LIN {X 0,Y 21.152,Z 455.053,A -85,B 0,C 180,E1 -30670.56,E2 -30670.56} C_VEL
LIN {X 0,Y 20.436,Z 453.143,A -85,B 0,C 180,E1 -30689.966,E2 -30689.966} C_VEL
LIN {X 0,Y 22.041,Z 449.239,A -85,B 0,C 180,E1 -30718.534,E2 -30718.534} C_VEL
LIN {X 0,Y 28.88,Z 443.167,A -85,B 0,C 180,E1 -30742.224,E2 -30742.224} C_VEL
LIN {X 0,Y 37.116,Z 436.479,A -85,B 0,C 180,E1 -30754.029,E2 -30754.029} C_VEL
LIN {X 0,Y 46.247,Z 428.101,A -85,B 0,C 180,E1 -30761.737,E2 -30761.737} C_VEL
LIN {X 0,Y 54.382,Z 419.589,A -85,B 0,C 180,E1 -30765.684,E2 -30765.684} C_VEL
LIN {X 0,Y 61.843,Z 410.185,A -85,B 0,C 180,E1 -30768.486,E2 -30768.486} C_VEL
LIN {X 0,Y 68.553,Z 399.902,A -85,B 0,C 180,E1 -30770.565,E2 -30770.565} C_VEL
LIN {X 0,Y 73.665,Z 390.513,A -85,B 0,C 180,E1 -30771.718,E2 -30771.718} C_VEL
LIN {X 0,Y 79.102,Z 377.77,A -85,B 0,C 180,E1 -30772.804,E2 -30772.804} C_VEL
LIN {X 0,Y 83.016,Z 365.075,A -85,B 0,C 180,E1 -30773.551,E2 -30773.551} C_VEL
LIN {X 0,Y 85.602,Z 351.961,A -85,B 0,C 180,E1 -30774.011,E2 -30774.011} C_VEL
LIN {X 0,Y 87.381,Z 337.149,A -85,B 0,C 180,E1 -30774.548,E2 -30774.548} C_VEL
LIN {X 0,Y 86.592,Z 333.719,A -85,B 0,C 180,E1 -30778.679,E2 -30778.679} C_VEL
LIN {X 0,Y 86.124,Z 331.369,A -85,B 0,C 180,E1 -30782.861,E2 -30782.861} C_VEL
LIN {X 0,Y 86.007,Z 330.813,A -85,B 0,C 180,E1 -30784.686,E2 -30784.686} C_VEL
LIN {X 0,Y 85.889,Z 330.908,A -85,B 0,C 180,E1 -30788.585,E2 -30788.585} C_VEL
LIN {X 0,Y 86.23,Z 332.513,A -85,B 0,C 180,E1 -30794.523,E2 -30794.523} C_VEL
LIN {X 0,Y 86.824,Z 335.034,A -85,B 0,C 180,E1 -30798.584,E2 -30798.584} C_VEL
LIN {X 0,Y 87.332,Z 337.027,A -85,B 0,C 180,E1 -30801.005,E2 -30801.005} C_VEL
LIN {X 0,Y 84.821,Z 355.596,A -85,B 0,C 180,E1 -30801.612,E2 -30801.612} C_VEL
LIN {X 0,Y 81.812,Z 368.186,A -85,B 0,C 180,E1 -30802.222,E2 -30802.222} C_VEL
LIN {X 0,Y 77.825,Z 379.916,A -85,B 0,C 180,E1 -30803.226,E2 -30803.226} C_VEL
LIN {X 0,Y 72.449,Z 391.692,A -85,B 0,C 180,E1 -30804.608,E2 -30804.608} C_VEL
LIN {X 0,Y 66.566,Z 401.881,A -85,B 0,C 180,E1 -30806.212,E2 -30806.212} C_VEL
LIN {X 0,Y 59.269,Z 412.386,A -85,B 0,C 180,E1 -30809.047,E2 -30809.047} C_VEL
LIN {X 0,Y 52.199,Z 420.784,A -85,B 0,C 180,E1 -30812.252,E2 -30812.252} C_VEL
LIN {X 0,Y 48.728,Z 424.445,A -85,B 0,C 180,E1 -30814.157,E2 -30814.157} C_VEL
LIN {X 0,Y 44.529,Z 428.33,A -85,B 0,C 180,E1 -30815.988,E2 -30815.988} C_VEL
LIN {X 0,Y 36.632,Z 434.249,A -85,B 0,C 180,E1 -30817.503,E2 -30817.503} C_VEL
LIN {X 0,Y 28.323,Z 439.531,A -85,B 0,C 180,E1 -30820.069,E2 -30820.069} C_VEL
LIN {X 0,Y 23.648,Z 442.421,A -85,B 0,C 180,E1 -30824.997,E2 -30824.997} C_VEL
LIN {X 0,Y 16.411,Z 447.259,A -85,B 0,C 180,E1 -30844.693,E2 -30844.693} C_VEL
LIN {X 0,Y 12.722,Z 451.395,A -85,B 0,C 180,E1 -30886.09,E2 -30886.09} C_VEL
LIN {X 0,Y 16.872,Z 454.463,A -85,B 0,C 180,E1 -30926.483,E2 -30926.483} C_VEL
LIN {X 0,Y 22.909,Z 456.047,A -85,B 0,C 180,E1 -30942.141,E2 -30942.141} C_VEL
LIN {X 0,Y 35.264,Z 457.62,A -85,B 0,C 180,E1 -30955.379,E2 -30955.379} C_VEL
LIN {X 0,Y 44.049,Z 457.774,A -85,B 0,C 180,E1 -30960.003,E2 -30960.003} C_VEL
LIN {X 0,Y 56.376,Z 456.921,A -85,B 0,C 180,E1 -30964.109,E2 -30964.109} C_VEL
LIN {X 0,Y 63.578,Z 455.839,A -85,B 0,C 180,E1 -30965.749,E2 -30965.749} C_VEL
LIN {X 0,Y 63.603,Z 455.843,A -85,B 0,C 180,E1 -30965.971,E2 -30965.971} C_VEL
LIN {X 0,Y 56.7,Z 457.023,A -85,B 0,C 180,E1 -30967.374,E2 -30967.374} C_VEL
LIN {X 0,Y 43.059,Z 458.202,A -85,B 0,C 180,E1 -30971.621,E2 -30971.621} C_VEL
LIN {X 0,Y 29.912,Z 457.897,A -85,B 0,C 180,E1 -30979.926,E2 -30979.926} C_VEL
LIN {X 0,Y 18.49,Z 456.019,A -85,B 0,C 180,E1 -31000.468,E2 -31000.468} C_VEL
LIN {X 0,Y 14.643,Z 454.496,A -85,B 0,C 180,E1 -31021.267,E2 -31021.267} C_VEL
LIN {X 0,Y 13.328,Z 452.539,A -85,B 0,C 180,E1 -31049.948,E2 -31049.948} C_VEL
LIN {X 0,Y 16.139,Z 448.54,A -85,B 0,C 180,E1 -31090.723,E2 -31090.723} C_VEL
LIN {X 0,Y 25.141,Z 442.314,A -85,B 0,C 180,E1 -31115.221,E2 -31115.221} C_VEL
LIN {X 0,Y 34.577,Z 435.505,A -85,B 0,C 180,E1 -31124.799,E2 -31124.799} C_VEL
LIN {X 0,Y 44.064,Z 427.412,A -85,B 0,C 180,E1 -31130.32,E2 -31130.32} C_VEL
LIN {X 0,Y 51.356,Z 420.152,A -85,B 0,C 180,E1 -31132.664,E2 -31132.664} C_VEL
LIN {X 0,Y 59.095,Z 410.986,A -85,B 0,C 180,E1 -31134.694,E2 -31134.694} C_VEL
LIN {X 0,Y 65.148,Z 402.341,A -85,B 0,C 180,E1 -31136.016,E2 -31136.016} C_VEL
LIN {X 0,Y 71.239,Z 391.903,A -85,B 0,C 180,E1 -31136.97,E2 -31136.97} C_VEL
LIN {X 0,Y 76.468,Z 380.436,A -85,B 0,C 180,E1 -31137.776,E2 -31137.776} C_VEL
LIN {X 0,Y 80.617,Z 368.351,A -85,B 0,C 180,E1 -31138.251,E2 -31138.251} C_VEL
LIN {X 0,Y 83.661,Z 355.3,A -85,B 0,C 180,E1 -31138.642,E2 -31138.642} C_VEL
LIN {X 0,Y 85.555,Z 341.204,A -85,B 0,C 180,E1 -31139.06,E2 -31139.06} C_VEL
LIN {X 0,Y 85.133,Z 338.175,A -85,B 0,C 180,E1 -31144.12,E2 -31144.12} C_VEL
LIN {X 0,Y 85.008,Z 337.862,A -85,B 0,C 180,E1 -31147.836,E2 -31147.836} C_VEL
LIN {X 0,Y 85.19,Z 339.365,A -85,B 0,C 180,E1 -31153.356,E2 -31153.356} C_VEL
LIN {X 0,Y 85.501,Z 341.237,A -85,B 0,C 180,E1 -31156.434,E2 -31156.434} C_VEL
LIN {X 0,Y 83.14,Z 357.34,A -85,B 0,C 180,E1 -31156.929,E2 -31156.929} C_VEL
LIN {X 0,Y 80.162,Z 369.125,A -85,B 0,C 180,E1 -31157.356,E2 -31157.356} C_VEL
LIN {X 0,Y 75.423,Z 382.156,A -85,B 0,C 180,E1 -31158.248,E2 -31158.248} C_VEL
LIN {X 0,Y 69.757,Z 393.773,A -85,B 0,C 180,E1 -31159.22,E2 -31159.22} C_VEL
LIN {X 0,Y 63.749,Z 403.615,A -85,B 0,C 180,E1 -31160.478,E2 -31160.478} C_VEL
LIN {X 0,Y 56.14,Z 413.877,A -85,B 0,C 180,E1 -31162.638,E2 -31162.638} C_VEL
LIN {X 0,Y 47.981,Z 422.846,A -85,B 0,C 180,E1 -31165.42,E2 -31165.42} C_VEL
LIN {X 0,Y 38.539,Z 431.46,A -85,B 0,C 180,E1 -31170.025,E2 -31170.025} C_VEL
LIN {X 0,Y 28.891,Z 438.849,A -85,B 0,C 180,E1 -31177.806,E2 -31177.806} C_VEL
LIN {X 0,Y 23.648,Z 442.421,A -85,B 0,C 180,E1 -31184.997,E2 -31184.997} C_VEL
LIN {X 0,Y 19.106,Z 445.129,A -85,B 0,C 180,E1 -31192.22,E2 -31192.22} C_VEL
LIN {X 0,Y 11.112,Z 448.972,A -85,B 0,C 180,E1 -31209.657,E2 -31209.657} C_VEL
LIN {X 0,Y 6.782,Z 451.6,A -85,B 0,C 180,E1 -31251.543,E2 -31251.543} C_VEL
LIN {X 0,Y 9.25,Z 453.584,A -85,B 0,C 180,E1 -31297.635,E2 -31297.635} C_VEL
LIN {X 0,Y 10.014,Z 453.798,A -85,B 0,C 180,E1 -31301.122,E2 -31301.122} C_VEL
LIN {X 0,Y 21.095,Z 456.424,A -85,B 0,C 180,E1 -31320.45,E2 -31320.45} C_VEL
LIN {X 0,Y 28.221,Z 457.431,A -85,B 0,C 180,E1 -31324.811,E2 -31324.811} C_VEL
LIN {X 0,Y 28.289,Z 457.473,A -85,B 0,C 180,E1 -31326.23,E2 -31326.23} C_VEL
LIN {X 0,Y 14.889,Z 455.504,A -85,B 0,C 180,E1 -31339.129,E2 -31339.129} C_VEL
LIN {X 0,Y 6.975,Z 452.963,A -85,B 0,C 180,E1 -31379.638,E2 -31379.638} C_VEL
LIN {X 0,Y 6.237,Z 451.907,A -85,B 0,C 180,E1 -31409.888,E2 -31409.888} C_VEL
LIN {X 0,Y 11.689,Z 447.806,A -85,B 0,C 180,E1 -31474.254,E2 -31474.254} C_VEL
LIN {X 0,Y 23.079,Z 441.464,A -85,B 0,C 180,E1 -31491.517,E2 -31491.517} C_VEL
LIN {X 0,Y 33.42,Z 434.531,A -85,B 0,C 180,E1 -31496.789,E2 -31496.789} C_VEL
LIN {X 0,Y 43.756,Z 425.966,A -85,B 0,C 180,E1 -31499.69,E2 -31499.69} C_VEL
LIN {X 0,Y 50.94,Z 418.881,A -85,B 0,C 180,E1 -31500.696,E2 -31500.696} C_VEL
LIN {X 0,Y 58.867,Z 409.462,A -85,B 0,C 180,E1 -31501.675,E2 -31501.675} C_VEL
LIN {X 0,Y 65.93,Z 399.161,A -85,B 0,C 180,E1 -31502.467,E2 -31502.467} C_VEL
LIN {X 0,Y 71.224,Z 389.754,A -85,B 0,C 180,E1 -31502.779,E2 -31502.779} C_VEL
LIN {X 0,Y 76.522,Z 377.784,A -85,B 0,C 180,E1 -31503.092,E2 -31503.092} C_VEL
LIN {X 0,Y 80.613,Z 365.216,A -85,B 0,C 180,E1 -31503.333,E2 -31503.333} C_VEL
LIN {X 0,Y 83.277,Z 352.696,A -85,B 0,C 180,E1 -31503.491,E2 -31503.491} C_VEL
LIN {X 0,Y 84.21,Z 345.881,A -85,B 0,C 180,E1 -31503.674,E2 -31503.674} C_VEL
